REGION Network 13: Check Pressure
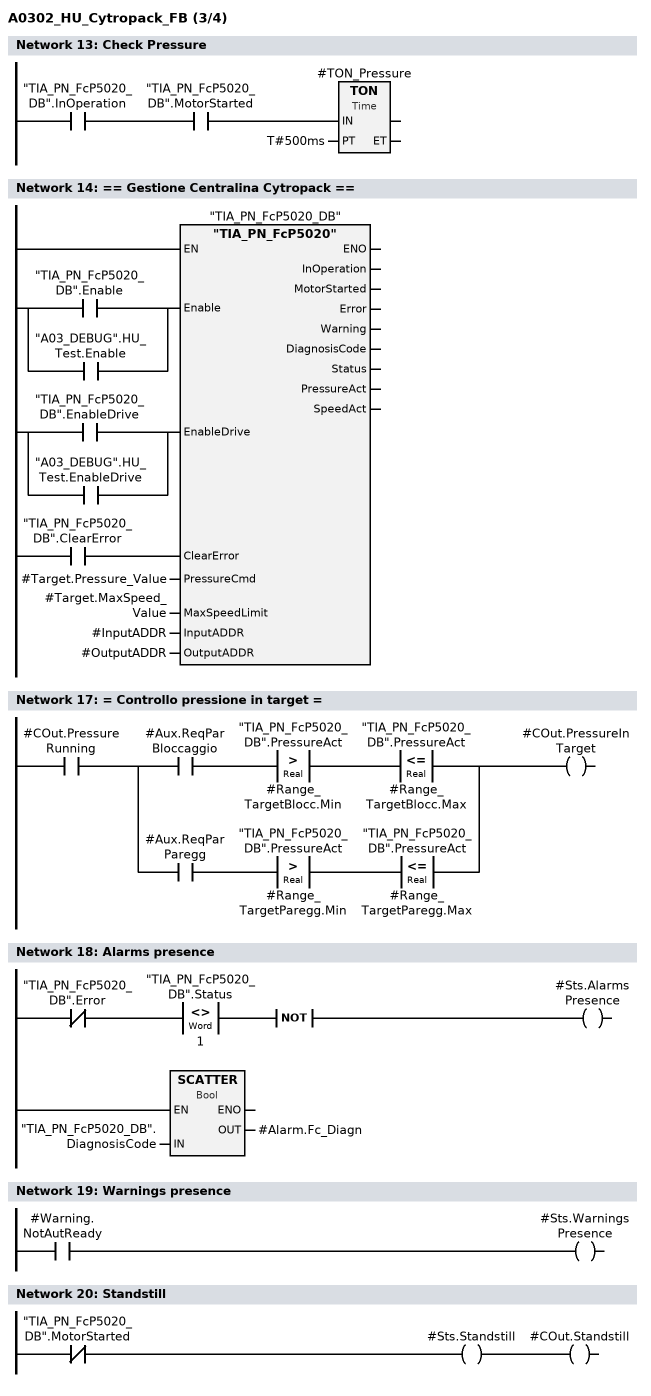
   RUNG wire#powerrail
      Contact( "TIA_PN_FcP5020_DB".InOperation )
      Contact( "TIA_PN_FcP5020_DB".MotorStarted )
      { S7_Templates := "time_type := Time" } #TON_Pressure.TON(pt := T#500ms, et =>)
   END_RUNG
   // the same network as SCL:
   #TON_Pressure.TON(IN := "TIA_PN_FcP5020_DB".InOperation AND "TIA_PN_FcP5020_DB".MotorStarted, PT := T#500ms);
END_REGION

REGION Network 14: == Gestione Centralina Cytropack ==
   RUNG wire#powerrail
      "TIA_PN_FcP5020_DB"(Enable := wire#w1, EnableDrive := wire#w2, ClearError := wire#w3, PressureCmd := #Target.Pressure_Value, MaxSpeedLimit := #Target.MaxSpeed_Value, InputADDR := #InputADDR, OutputADDR := #OutputADDR, InOperation =>, MotorStarted =>, Error =>, Warning =>, DiagnosisCode =>, Status =>, PressureAct =>, SpeedAct =>)
   END_RUNG
   RUNG wire#powerrail
      Contact( "TIA_PN_FcP5020_DB".Enable )
   END_RUNG wire#w1
   RUNG wire#powerrail
      Contact( "A03_DEBUG".HU_Test.Enable )
   END_RUNG wire#w1
   RUNG wire#powerrail
      Contact( "TIA_PN_FcP5020_DB".EnableDrive )
   END_RUNG wire#w2
   RUNG wire#powerrail
      Contact( "A03_DEBUG".HU_Test.EnableDrive )
   END_RUNG wire#w2
   RUNG wire#powerrail
      Contact( "TIA_PN_FcP5020_DB".ClearError )
   END_RUNG wire#w3
   // the same network as SCL:
   "TIA_PN_FcP5020_DB"(Enable := "TIA_PN_FcP5020_DB".Enable OR "A03_DEBUG".HU_Test.Enable,   // "TIA_PN_FcP5020"
                       EnableDrive := "TIA_PN_FcP5020_DB".EnableDrive OR "A03_DEBUG".HU_Test.EnableDrive,
                       ClearError := "TIA_PN_FcP5020_DB".ClearError,
                       PressureCmd := #Target.Pressure_Value,
                       MaxSpeedLimit := #Target.MaxSpeed_Value,
                       InputADDR := #InputADDR,
                       OutputADDR := #OutputADDR);
END_REGION

REGION Network 16: <<< MACHINE STATUS >>>
END_REGION

REGION Network 17: = Controllo pressione in target =
   RUNG wire#powerrail
      Contact( #COut.PressureRunning )
      wire#w1
      Contact( #Aux.ReqParBloccaggio )
      { S7_Templates := "SrcType := Real" } GT_Contact(in1 := "TIA_PN_FcP5020_DB".PressureAct, in2 := #Range_TargetBlocc.Min)
      { S7_Templates := "SrcType := Real" } LE_Contact(in1 := "TIA_PN_FcP5020_DB".PressureAct, in2 := #Range_TargetBlocc.Max)
      wire#w2
      Coil( #COut.PressureInTarget )
   END_RUNG
   RUNG wire#w1
      Contact( #Aux.ReqParParegg )
      { S7_Templates := "SrcType := Real" } GT_Contact(in1 := "TIA_PN_FcP5020_DB".PressureAct, in2 := #Range_TargetParegg.Min)
      { S7_Templates := "SrcType := Real" } LE_Contact(in1 := "TIA_PN_FcP5020_DB".PressureAct, in2 := #Range_TargetParegg.Max)
   END_RUNG wire#w2
   // the same network as SCL:
   #COut.PressureInTarget := #COut.PressureRunning AND ((#Aux.ReqParBloccaggio AND ("TIA_PN_FcP5020_DB".PressureAct > #Range_TargetBlocc.Min) AND ("TIA_PN_FcP5020_DB".PressureAct <= #Range_TargetBlocc.Max)) OR (#Aux.ReqParParegg AND ("TIA_PN_FcP5020_DB".PressureAct > #Range_TargetParegg.Min) AND ("TIA_PN_FcP5020_DB".PressureAct <= #Range_TargetParegg.Max)));
END_REGION

REGION Network 18: Alarms presence
   RUNG wire#powerrail
      I_Contact( "TIA_PN_FcP5020_DB".Error )
      { S7_Templates := "SrcType := Word" } NE_Contact(in1 := "TIA_PN_FcP5020_DB".Status, in2 := 1)
      Not()
      Coil( #Sts.AlarmsPresence )
   END_RUNG
   RUNG wire#powerrail
      { S7_Templates := "[dest_type := Bool, src_type := Word]" } SCATTER(IN := "TIA_PN_FcP5020_DB".DiagnosisCode, OUT => #Alarm.Fc_Diagn)
   END_RUNG
   // the same network as SCL:
   #Sts.AlarmsPresence := NOT (NOT "TIA_PN_FcP5020_DB".Error AND ("TIA_PN_FcP5020_DB".Status <> 1));
   SCATTER(IN := "TIA_PN_FcP5020_DB".DiagnosisCode, OUT => #Alarm.Fc_Diagn);
END_REGION

REGION Network 19: Warnings presence
   RUNG wire#powerrail
      Contact( #Warning.NotAutReady )
      Coil( #Sts.WarningsPresence )
   END_RUNG
   // the same network as SCL:
   #Sts.WarningsPresence := #Warning.NotAutReady;
END_REGION

REGION Network 20: Standstill
   RUNG wire#powerrail
      I_Contact( "TIA_PN_FcP5020_DB".MotorStarted )
      Coil( #Sts.Standstill )
      Coil( #COut.Standstill )
   END_RUNG
   // the same network as SCL:
   #Sts.Standstill := NOT "TIA_PN_FcP5020_DB".MotorStarted;
   #COut.Standstill := NOT "TIA_PN_FcP5020_DB".MotorStarted;
END_REGION

REGION Network 21: Stop for aborting
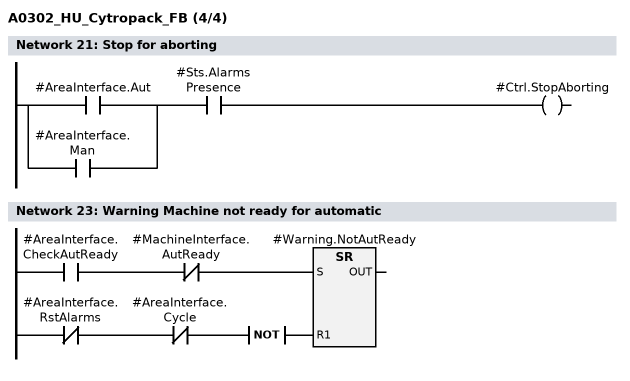
   RUNG wire#powerrail
      Contact( #AreaInterface.Aut )
      wire#w1
      Contact( #Sts.AlarmsPresence )
      Coil( #Ctrl.StopAborting )
   END_RUNG
   RUNG wire#powerrail
      Contact( #AreaInterface.Man )
   END_RUNG wire#w1
   // the same network as SCL:
   #Ctrl.StopAborting := (#AreaInterface.Aut OR #AreaInterface.Man) AND #Sts.AlarmsPresence;
END_REGION

REGION Network 22 (SCL): Collect machine to zone interface

   #MachineInterface.AutReady := #AreaInterface.Aut AND NOT #Sts.AlarmsPresence;
   #MachineInterface.Aborting := #Ctrl.StopAborting;
   #MachineInterface.MotionsStandStill := #TON_NoPendingCmd.Q AND #Sts.Standstill;
   #MachineInterface.AckStopInPhase := #Ctrl.StopInPhase  AND #MachineInterface.MotionsStandStill;
   #MachineInterface.AckStopProgrammed := #Ctrl.StopProgrammed AND #MachineInterface.MotionsStandStill;
   #MachineInterface.AlarmsPresence := #Sts.AlarmsPresence;
   #MachineInterface.WarningPresence := #Sts.WarningsPresence;
END_REGION

REGION Network 23: Warning Machine not ready for automatic
   RUNG wire#powerrail
      Contact( #AreaInterface.CheckAutReady )
      I_Contact( #MachineInterface.AutReady )
      S_SR(operand := #Warning.NotAutReady, r1 := wire#w1)
   END_RUNG
   RUNG wire#powerrail
      I_Contact( #AreaInterface.RstAlarms )
      I_Contact( #AreaInterface.Cycle )
      Not()
   END_RUNG wire#w1
   // the same network as SCL:
   IF #AreaInterface.CheckAutReady AND NOT #MachineInterface.AutReady THEN
       #Warning.NotAutReady := TRUE;   // SR flip-flop
   END_IF;
   IF NOT (NOT #AreaInterface.RstAlarms AND NOT #AreaInterface.Cycle) THEN
       #Warning.NotAutReady := FALSE;
   END_IF;
END_REGION

REGION Network 24 (SCL): Return value variable
   (* LBO TEST
   // Read data from EFC's PROFINET input area
   #iReturnVal := DPRD_DAT(LADDR := #InputADDR, RECORD => #stInputData);
   // Read data failed
   IF (#iReturnVal <> 0) THEN
       #Error := TRUE;
       #bFBErrorDPRD_DPWR := TRUE;
       RETURN;
   END_IF;
   *)
END_REGION
END_FUNCTION_BLOCK

FUNCTION "A0302_Spintore_CALL" : Void   // FC1, LAD
// stored: SetENOAutomatically false
   VAR_TEMP
      Missing_Input : Bool;
      Missing_Output : Bool;
   END_VAR
   VAR CONSTANT
      MISSING : Int;
   END_VAR
BEGIN

REGION Network 1 (SCL): << TRASFERIMENTO stati CIn del blocco >>
   REGION TRASFERIMENTO CIn MANAGER
       "A0302_Spintore".Cin.Manager := "A0302_Manager".COut.SpintoreLong;
       //
       "A0302_Spintore".Cin.SemiAut_Pb := "A0302_Manager".DataIn.SemiAut_Pb;

   END_REGION ;

   REGION TRASFERIMENTO BORDATRICE
       "A0302_Spintore".Cin.Bordatrice.Ax := "A0302_Bordatrice".COut.Ax;
       "A0302_Spintore".Cin.Bordatrice.Sens.FTC_Uscita := "A0302_Bordatrice".IEC_FTC_UscitaBordatrice.FTC_On;
       "A0302_Spintore".Cin.Bordatrice.Perc_Vel := 50.0;
       "A0302_Spintore".Cin.Bordatrice.TargetVel := "A0302_Bordatrice".COut.Ax.ActualVelocity;

   END_REGION ;

   REGION TRASFERIMENTO CIn FERMI P4
       "A0302_Spintore".Cin.P4.Fermi := "A0301_Fermi_P4".COut.Fermi;
   END_REGION ;

   REGION TRASFERIMENTO SPINTORI LATERALI CIn P5
       "A0302_Spintore".Cin.P5.Spintore_Lat.Spin_Lat1 := "A0301_Spintore_Lat".COut.Spin_Lat1;
       "A0302_Spintore".Cin.P5.Spintore_Lat.Spin_Lat2 := "A0301_Spintore_Lat".COut.Spin_Lat2;
       "A0302_Spintore".Cin.P5."En/Dis_SpinLat_2" := "A0301_Spintore_Lat".Sts."En/Dis_SpinLat_2";
       "A0302_Spintore".Cin.P5.QuotaIngombro_SpinLat2 := "PrjConfig_A03".A0301.SpintoreLaterale.QuotaIngombro_SpinLat2;
       "A0302_Spintore".Cin.P5.QuotaIngombro_SpinLat1 := "PrjConfig_A03".A0301.SpintoreLaterale.QuotaIngombro_SpinLat1;

   END_REGION ;

   REGION TRASFERIMENTO CIn TRASPORTO 
       // Trasferimenti status lettura posizioni Trasporto al Cin delle stazioni
       "A0302_Spintore".Cin.Trasporto := "A0301_Trasporto".COut.Ax;
   END_REGION ;
END_REGION

REGION Network 2 (SCL): << TRASFERIMENTO stati DataIn >>
   REGION TRASFERIMENTO #DataIn STATI OPERATION BUTTON STAZIONE SPINTORE LATERALE 
       // PB FERMI VERTICALI
       "A0302_Spintore".DataIn.OP.Rest := "A03_HMI".MB3.Button.A0302.SpintoreLong.OP.Rest;
       "A0302_Spintore".DataIn.OP.Work := "A03_HMI".MB3.Button.A0302.SpintoreLong.OP.Work;
   END_REGION ;

   REGION TRASFERIMENTO STATO LETTURA SENSORI SPINTORE 

       "A0302_Spintore".DataIn.P5.Orz_AnalSens := "A0302_AI_Ammortizatore_Posizionamento";
       "A0302_Spintore".DataIn.P5.FTC_FuoriIngombro_A0301 := "A0302_Bordatrice_Banco_4_Lato_1_Phc_AtEntry";

   END_REGION ;
END_REGION

REGION Network 3: << DataIn Ax - Asse Spintore pezzo >>
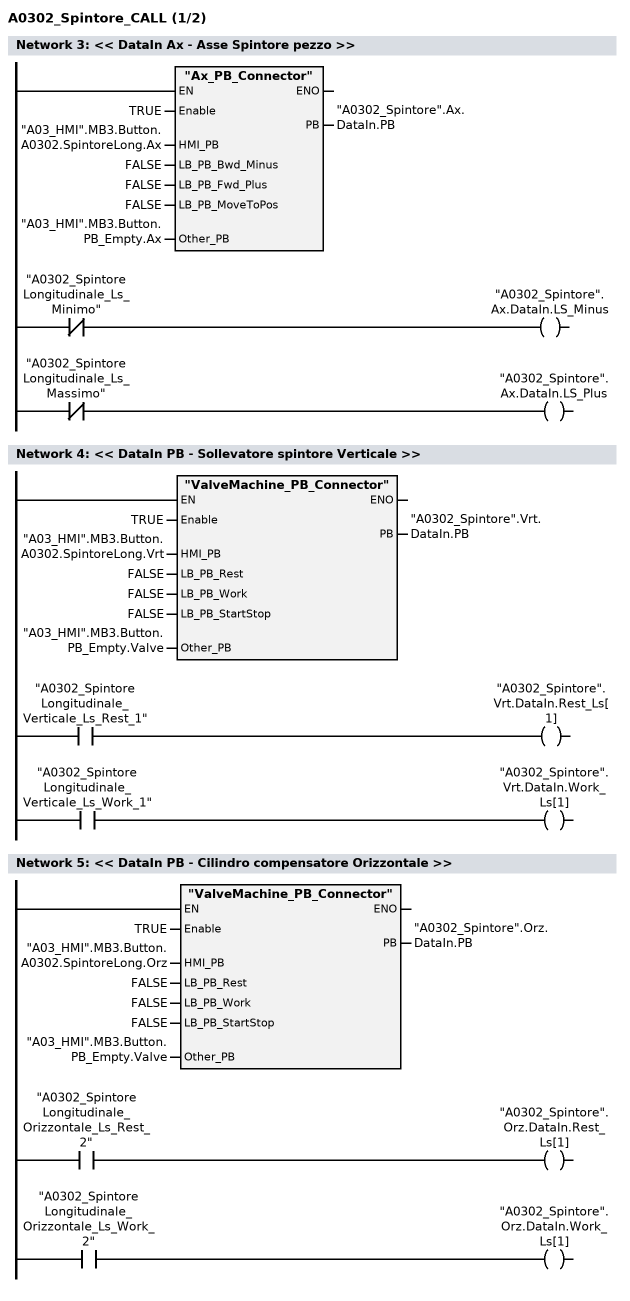
   RUNG wire#powerrail
      "Ax_PB_Connector"(Enable := TRUE, HMI_PB := "A03_HMI".MB3.Button.A0302.SpintoreLong.Ax, LB_PB_Bwd_Minus := FALSE, LB_PB_Fwd_Plus := FALSE, LB_PB_MoveToPos := FALSE, Other_PB := "A03_HMI".MB3.Button.PB_Empty.Ax, PB => "A0302_Spintore".Ax.DataIn.PB)
   END_RUNG
   RUNG wire#powerrail
      I_Contact( "A0302_SpintoreLongitudinale_Ls_Minimo" )
      Coil( "A0302_Spintore".Ax.DataIn.LS_Minus )
   END_RUNG
   RUNG wire#powerrail
      I_Contact( "A0302_SpintoreLongitudinale_Ls_Massimo" )
      Coil( "A0302_Spintore".Ax.DataIn.LS_Plus )
   END_RUNG
   // the same network as SCL:
   "Ax_PB_Connector"(Enable := TRUE,
                     HMI_PB := "A03_HMI".MB3.Button.A0302.SpintoreLong.Ax,
                     LB_PB_Bwd_Minus := FALSE,
                     LB_PB_Fwd_Plus := FALSE,
                     LB_PB_MoveToPos := FALSE,
                     Other_PB := "A03_HMI".MB3.Button.PB_Empty.Ax,
                     PB => "A0302_Spintore".Ax.DataIn.PB);
   "A0302_Spintore".Ax.DataIn.LS_Minus := NOT "A0302_SpintoreLongitudinale_Ls_Minimo";
   "A0302_Spintore".Ax.DataIn.LS_Plus := NOT "A0302_SpintoreLongitudinale_Ls_Massimo";
END_REGION

REGION Network 4: << DataIn PB - Sollevatore spintore Verticale >>
   RUNG wire#powerrail
      "ValveMachine_PB_Connector"(Enable := TRUE, HMI_PB := "A03_HMI".MB3.Button.A0302.SpintoreLong.Vrt, LB_PB_Rest := FALSE, LB_PB_Work := FALSE, LB_PB_StartStop := FALSE, Other_PB := "A03_HMI".MB3.Button.PB_Empty.Valve, PB => "A0302_Spintore".Vrt.DataIn.PB)
   END_RUNG
   RUNG wire#powerrail
      Contact( "A0302_SpintoreLongitudinale_Verticale_Ls_Rest_1" )
      Coil( "A0302_Spintore".Vrt.DataIn.Rest_Ls[1] )
   END_RUNG
   RUNG wire#powerrail
      Contact( "A0302_SpintoreLongitudinale_Verticale_Ls_Work_1" )
      Coil( "A0302_Spintore".Vrt.DataIn.Work_Ls[1] )
   END_RUNG
   // the same network as SCL:
   "ValveMachine_PB_Connector"(Enable := TRUE,
                           HMI_PB := "A03_HMI".MB3.Button.A0302.SpintoreLong.Vrt,
                           LB_PB_Rest := FALSE,
                           LB_PB_Work := FALSE,
                           LB_PB_StartStop := FALSE,
                           Other_PB := "A03_HMI".MB3.Button.PB_Empty.Valve,
                           PB => "A0302_Spintore".Vrt.DataIn.PB);
   "A0302_Spintore".Vrt.DataIn.Rest_Ls[1] := "A0302_SpintoreLongitudinale_Verticale_Ls_Rest_1";
   "A0302_Spintore".Vrt.DataIn.Work_Ls[1] := "A0302_SpintoreLongitudinale_Verticale_Ls_Work_1";
END_REGION

REGION Network 5: << DataIn PB - Cilindro compensatore Orizzontale >>
   RUNG wire#powerrail
      "ValveMachine_PB_Connector"(Enable := TRUE, HMI_PB := "A03_HMI".MB3.Button.A0302.SpintoreLong.Orz, LB_PB_Rest := FALSE, LB_PB_Work := FALSE, LB_PB_StartStop := FALSE, Other_PB := "A03_HMI".MB3.Button.PB_Empty.Valve, PB => "A0302_Spintore".Orz.DataIn.PB)
   END_RUNG
   RUNG wire#powerrail
      Contact( "A0302_SpintoreLongitudinale_Orizzontale_Ls_Rest_2" )
      Coil( "A0302_Spintore".Orz.DataIn.Rest_Ls[1] )
   END_RUNG
   RUNG wire#powerrail
      Contact( "A0302_SpintoreLongitudinale_Orizzontale_Ls_Work_2" )
      Coil( "A0302_Spintore".Orz.DataIn.Work_Ls[1] )
   END_RUNG
   // the same network as SCL:
   "ValveMachine_PB_Connector"(Enable := TRUE,
                           HMI_PB := "A03_HMI".MB3.Button.A0302.SpintoreLong.Orz,
                           LB_PB_Rest := FALSE,
                           LB_PB_Work := FALSE,
                           LB_PB_StartStop := FALSE,
                           Other_PB := "A03_HMI".MB3.Button.PB_Empty.Valve,
                           PB => "A0302_Spintore".Orz.DataIn.PB);
   "A0302_Spintore".Orz.DataIn.Rest_Ls[1] := "A0302_SpintoreLongitudinale_Orizzontale_Ls_Rest_2";
   "A0302_Spintore".Orz.DataIn.Work_Ls[1] := "A0302_SpintoreLongitudinale_Orizzontale_Ls_Work_2";
END_REGION

REGION Network 6 (SCL): DSI
   //
   "A0302_Spintore".DSI_Feed := "F_DB".DSI_Spintore;
   "A0302_Spintore".DSI_Valve := "F_DB".DSI_V_Air_A0301_A0302;
END_REGION

REGION Network 7 (SCL): HW
   "A0302_Spintore".HWID_Ax_TEL111 := "HW_Const_Values".CU5_PN_1560A1_2_Standard_telegram_1_2;
END_REGION

REGION Network 8 (SCL): Drive
   //
   "A0302_Spintore".Drive.Infeed_ON := "Areas_ITF".AG.Infeed_Running;
   "A0302_Spintore".Drive.AccessPoint :=  "HW_Const_Values".CU5_PN_600A1_ModuleAccessPoint;
   "A0302_Spintore".Drive.AxisID := "CU5_ID_6_1560A1_2_1600M1";
   "A0302_Spintore".Drive.TokenChain := "TOKENCHAIN_CU5";
END_REGION

REGION Network 9: [Spintore Longitudinale] - Machine Call
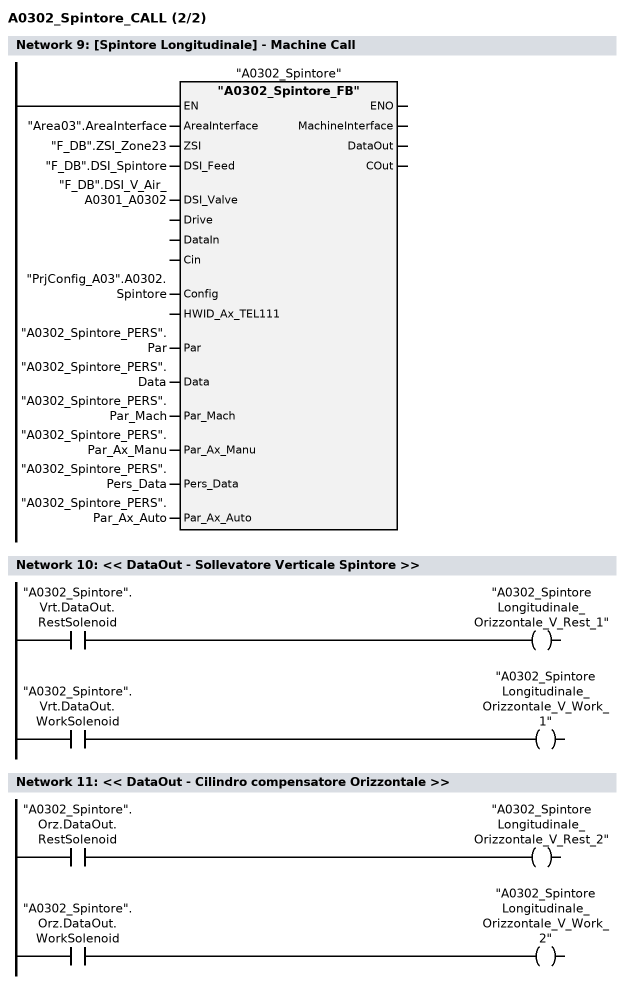
   RUNG wire#powerrail
      "A0302_Spintore"(AreaInterface := "Area03".AreaInterface, ZSI := "F_DB".ZSI_Zone23, DSI_Feed := "F_DB".DSI_Spintore, DSI_Valve := "F_DB".DSI_V_Air_A0301_A0302, Drive :=, DataIn :=, Cin :=, Config := "PrjConfig_A03".A0302.Spintore, HWID_Ax_TEL111 :=, Par := "A0302_Spintore_PERS".Par, Data := "A0302_Spintore_PERS".Data, Par_Mach := "A0302_Spintore_PERS".Par_Mach, Par_Ax_Manu := "A0302_Spintore_PERS".Par_Ax_Manu, Pers_Data := "A0302_Spintore_PERS".Pers_Data, Par_Ax_Auto := "A0302_Spintore_PERS".Par_Ax_Auto, MachineInterface =>, DataOut =>, COut =>)
   END_RUNG
   // the same network as SCL:
   "A0302_Spintore"(AreaInterface := "Area03".AreaInterface,   // "A0302_Spintore_FB"
                    ZSI := "F_DB".ZSI_Zone23,
                    DSI_Feed := "F_DB".DSI_Spintore,
                    DSI_Valve := "F_DB".DSI_V_Air_A0301_A0302,
                    Config := "PrjConfig_A03".A0302.Spintore,
                    Par := "A0302_Spintore_PERS".Par,
                    Data := "A0302_Spintore_PERS".Data,
                    Par_Mach := "A0302_Spintore_PERS".Par_Mach,
                    Par_Ax_Manu := "A0302_Spintore_PERS".Par_Ax_Manu,
                    Pers_Data := "A0302_Spintore_PERS".Pers_Data,
                    Par_Ax_Auto := "A0302_Spintore_PERS".Par_Ax_Auto);
END_REGION

REGION Network 10: << DataOut - Sollevatore Verticale Spintore >>
   RUNG wire#powerrail
      Contact( "A0302_Spintore".Vrt.DataOut.RestSolenoid )
      Coil( "A0302_SpintoreLongitudinale_Orizzontale_V_Rest_1" )
   END_RUNG
   RUNG wire#powerrail
      Contact( "A0302_Spintore".Vrt.DataOut.WorkSolenoid )
      Coil( "A0302_SpintoreLongitudinale_Orizzontale_V_Work_1" )
   END_RUNG
   // the same network as SCL:
   "A0302_SpintoreLongitudinale_Orizzontale_V_Rest_1" := "A0302_Spintore".Vrt.DataOut.RestSolenoid;
   "A0302_SpintoreLongitudinale_Orizzontale_V_Work_1" := "A0302_Spintore".Vrt.DataOut.WorkSolenoid;
END_REGION

REGION Network 11: << DataOut - Cilindro compensatore Orizzontale >>
   RUNG wire#powerrail
      Contact( "A0302_Spintore".Orz.DataOut.RestSolenoid )
      Coil( "A0302_SpintoreLongitudinale_Orizzontale_V_Rest_2" )
   END_RUNG
   RUNG wire#powerrail
      Contact( "A0302_Spintore".Orz.DataOut.WorkSolenoid )
      Coil( "A0302_SpintoreLongitudinale_Orizzontale_V_Work_2" )
   END_RUNG
   // the same network as SCL:
   "A0302_SpintoreLongitudinale_Orizzontale_V_Rest_2" := "A0302_Spintore".Orz.DataOut.RestSolenoid;
   "A0302_SpintoreLongitudinale_Orizzontale_V_Work_2" := "A0302_Spintore".Orz.DataOut.WorkSolenoid;
END_REGION
END_FUNCTION

FUNCTION_BLOCK "A0302_Spintore_FB"   // FB91, LAD
// stored: MemoryReserve 100, SetENOAutomatically false
   VAR_INPUT
      AreaInterface : "AreaInterface";
      ZSI : "udt_ZoneSafetyInterface";
      DSI_Feed : "udt_DeviceSafetyInterface";
      DSI_Valve : "udt_DeviceSafetyInterface";
      Drive : "TAx_DriveInterface";
      DataIn : Struct
         OP : "OP_PB";
         P5 { ExternalAccessible := 'False'; ExternalVisible := 'False'; ExternalWritable := 'False'} : Struct
            Orz_AnalSens : Int;
            FTC_FuoriIngombro_A0301 : Bool;   // FTC fuori ingombro lato bordatrice
         END_STRUCT;
      END_STRUCT;
      Cin : Struct
         Manager { ExternalWritable := 'False'} : Struct
            EnableStopDoorOpeningReq : Bool;
            EnableStopInPhase : Bool;
            EnableStopProgrammed : Bool;
            Control_ON : Bool;
            REST_Req : Bool;
            WORK_Req : Bool;
            Rest : Bool;
            Work : Bool;
         END_STRUCT;
         SemiAut_Pb { ExternalAccessible := 'False'; ExternalVisible := 'False'; ExternalWritable := 'False'} : Bool;
         P4 { ExternalWritable := 'False'} : Struct
            Fermi : "ValveMachine_COut";
         END_STRUCT;
         P5 { ExternalWritable := 'False'} : Struct
            "En/Dis_SpinLat_2" : Bool;   // 1=Enable / 0=Disable
            QuotaIngombro_SpinLat2 : Real;
            QuotaIngombro_SpinLat1 : Real;
            Spintore_Lat : Struct
               Spin_Lat1 : Struct
                  Standstill : Bool;
                  Rest_CheckNext : Bool;
                  Work_CheckNext : Bool;
                  Rest : Bool;
                  Work : Bool;
               END_STRUCT;
               Spin_Lat2 : Struct
                  Standstill : Bool;
                  Rest_CheckNext : Bool;
                  Work_CheckNext : Bool;
                  Rest : Bool;
                  Work : Bool;
               END_STRUCT;
               Vrt_1 : "ValveMachine_COut";
               Orz_1 : "ValveMachine_COut";
               Vrt_2 : "ValveMachine_COut";
               Orz_2 : "ValveMachine_COut";
               Sollevatori : "ValveMachine_COut";
            END_STRUCT;
         END_STRUCT;
         Trasporto { ExternalAccessible := 'False'; ExternalVisible := 'False'; ExternalWritable := 'False'} : "SpeedMachine_COut";
         Bordatrice : Struct   // *************************
            Ax : "Positioning_EPOS_Machine_COut";
            TargetVel : LReal;
            Perc_Vel : LReal;
            Sens : Struct
               FTC_Uscita : Bool;
            END_STRUCT;
         END_STRUCT;
      END_STRUCT;
      Config : Struct
         Ax : "Positioning_EPOS_Machine_Config_NEW";
         Vrt : "ValveMachine_Config";
         Orz : "ValveMachine_Config";
         SpintoreLat : Struct
            QuotaIngombro_SpinLat2 : Real := 2705.0;
            QuotaIngombro_SpinLat1 : Real := 4777.0;
         END_STRUCT;
         Bordatrice : Struct
            QuotaIngresso : Real := 600.0;
         END_STRUCT;
         DelayMissingCondition : Time;
      END_STRUCT;
      HWID_Ax_TEL111 : HW_SUBMODULE;
   END_VAR
   VAR_OUTPUT
      MachineInterface : "MachineInterface";
      DataOut : "Positioning_EPOS_Machine_DataOut";
      COut : Struct
         Ax_Sts : Struct
            PosAttesa_Reached : Bool;
            PosFineSpinta_Reached : Bool;
         END_STRUCT;
         Ax : "Positioning_EPOS_Machine_COut";
         Spintore : "ValveMachine_COut";
         Vrt : "ValveMachine_COut";
         Orz : "ValveMachine_COut";
      END_STRUCT;
   END_VAR
   VAR_IN_OUT
      Par : Struct
         Sens : "Analogic_SensorManagement_Par";
      END_STRUCT;
      Data : Struct
         Sens : "Analogic_SensorManagement_Data";
         HMI : "HMI_Preset";
         Ax_Pos : "A0301_Mach_Ax_Pos_Data";
      END_STRUCT;
      Par_Mach : "A0301_Mach_Sens_Par";
      Par_Ax_Manu : "Positioning_EPOS_Machine_Par";
      Pers_Data : Struct
         EncoderAbsolute_Preset_OK : Bool;
         Persistent_ActualPosition : LReal;
      END_STRUCT;
      Par_Ax_Auto : "A0301_Mach_Speed_Par";
   END_VAR
   VAR
      Alarm : Struct
         Ax : "Positioning_EPOS_Machine_Alr";
         Ax_NeedPreset { S7_SetPoint := 'True'} : Bool;
         Vrt : "ValveAlr";
         Orz : "ValveAlr";
         Orz_AnalSens_Issue : Bool;
         Orz_AnalSens_Compressed : Bool;
      END_STRUCT;
      Warning : Struct
         Ax : "Positioning_EPOS_Machine_Wng";
         Vrt : "ValveMachine_Wng";
         Orz { S7_SetPoint := 'True'} : "ValveMachine_Wng";
         Orz_AnalSens { S7_SetPoint := 'True'} : "Analogic_SensorManagement_Warning";
         OP_REST_MissingCnd : Bool;   // Mancanza comando arresto
         OP_WORK_MissingCnd : Bool;   // Mancanza consenso lavoro
      END_STRUCT;
      Sts : Struct
         ReadyForMove : Bool;   // Pronto al movimento
         OP_CanMoveFreely : Bool;
         OP_Ax_Rest_Cnd : Bool;
         OP_Ax_Work_Cnd : Bool;
         OP_Spin_Rest_Cnd : Bool;
         OP_Spin_Work_Cnd : Bool;
         A0301_Beam_BLean : Real;
         A0302_Beam_BLean : Real;
         Vrt_Work_ExtEnable : Bool;
         Orz_Work_ExtEnable : Bool;
      END_STRUCT;
      Ctrl : Struct
         SpinVrtOrz : Struct
            OP_Rest_Man : Bool;
            OP_Work_Man : Bool;
            OP_Rest_Aut : Bool;
            OP_Work_Aut : Bool;
            OP_Rest : Bool;
            OP_Work : Bool;
         END_STRUCT;
         Ax : Struct
            OP_Rest_Man : Bool;
            OP_Work_Man : Bool;
            OP_Rest_Aut : Bool;
            OP_Work_Aut : Bool;
            OP_Rest : Bool;
            OP_Work : Bool;
            Vel : LReal;
            VelMax : Real;
            Dec : LReal;
         END_STRUCT;
      END_STRUCT;
      HMI : Struct
         Ax : "AnalogSens_HmiData";
         Orz_AnalSens_PB_Preset { ExternalAccessible := 'False'; ExternalVisible := 'False'; ExternalWritable := 'False'} : Bool;   // Pulsante Preset value
         Orz_AnalSens_Preset_Value : LReal;
      END_STRUCT;
      Ax { S7_SetPoint := 'True'} : "Positioning_EPOS_Machine_FB_NEW";   // Spintore longitudinale
      Vrt { S7_SetPoint := 'True'} : "ValveMachine_FB";   // Sollevatore verticale
      Orz { S7_SetPoint := 'True'} : "ValveMachine_FB";   // Compensatore orizzontale
      Orz_AnalSens { S7_SetPoint := 'True'} : "Analogic_SensorManagement";
      ValueBLeanOvr : Array[1..15] of Real;
      IEC : Struct
         TON_DelayFTC_Ingombro_A0301 : IEC_TIMER;
         TOF_DelayFTC_Ingombro_A0301 { S7_SetPoint := 'True'} : IEC_TIMER;
         FTC_On { S7_SetPoint := 'True'} : Bool;
      END_STRUCT;
      AUX : Struct
         OP_Rest_PB : Bool;
         OP_Work_PB : Bool;
      END_STRUCT;
      TON_OP_REST_MissingCnd { S7_SetPoint := 'True'} : TON_TIME;
      TON_OP_WORK_MissingCnd { S7_SetPoint := 'True'} : TON_TIME;
      BTrk_Item : Struct
         BLean : Real;
         O_ID : DInt;
      END_STRUCT;
   END_VAR
   VAR_TEMP
      i : Int;
      DecMax : LReal;
      Orz_SpazioSafe : LReal;
      Calcoli : Struct
         SUB_SpinLat2 : LReal;
         SUB_SpinLat1 : LReal;
         Pos_Target_2 : LReal;
         Pos_Target_1 : LReal;
         Ax_Target : LReal;
      END_STRUCT;
      PE : Struct
         OP_Rest_PB : Bool;
         OP_Work_PB : Bool;
      END_STRUCT;
      BTrk_GetData_A0302 : Struct
         indx : Int;   // Se trovato tra i TODO / ENDING / OUT questo è l'indice dove sono stati prelevati i dati
         Sts : Int;   // 0 = Non Trovato; 0 = ACT; 1 = TODO; 2=ENDING; 3 = OUT
         Item : "Prod_Item_small";
      END_STRUCT;
      BTrk_GetData_A0301 : Struct
         indx : Int;   // Se trovato tra i TODO / ENDING / OUT questo è l'indice dove sono stati prelevati i dati
         Sts : Int;   // 0 = Non Trovato; 0 = ACT; 1 = TODO; 2=ENDING; 3 = OUT
         Item : "Prod_Item_small";
      END_STRUCT;
      Stop_Ax_SpinLong : Bool;
      GetData_A0301_B : Bool;
      GetData_A0302_In : Bool;
   END_VAR
   VAR CONSTANT
      Offset_SpinLong_To_SpinLat2 : Real;   // Offset calcolato da quota ingombro Spintore Laterale2 per bloccare Spintore Longitudinale e allarme se SpinLat2 alto
      Offset_SpinLong_To_SpinLat1 : Real;   // Offset calcolato da quota ingombro Spintore Laterale1 per bloccare Spintore Longitudinale e allarme se SpinLat1 alto
   END_VAR
   // Orz_AnalSens.Filter.Tau := T#10ms;
   VAR_TEMP   // added for the SCL form of the ladder/FBD networks
      _w1 : Bool;
      _w2 : Bool;
      _w3 : Bool;
      _w4 : Bool;
      _w5 : Bool;
      _w6 : Bool;
   END_VAR
BEGIN

REGION Network 1 (SCL): Reset allarmi
   IF #AreaInterface.RstAlarms THEN
       #Alarm.Orz_AnalSens_Issue := FALSE;
       #Warning.Orz_AnalSens.SignalError := FALSE;
   END_IF;
END_REGION

REGION Network 2: <+>
END_REGION

REGION Network 4: CONTROLLO MES lunghezza Beams
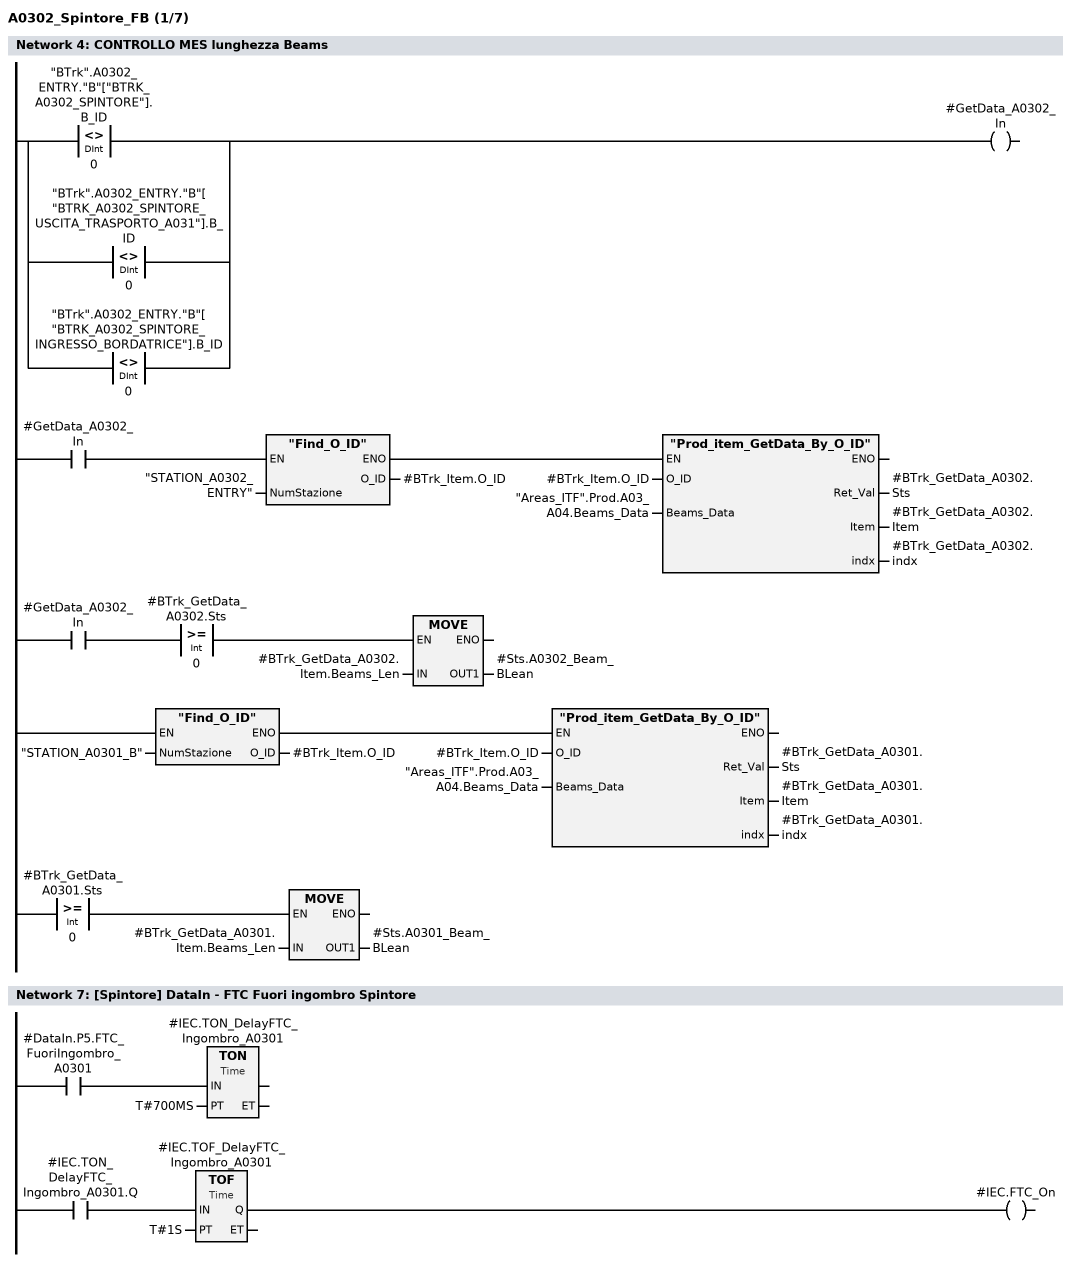
   RUNG wire#powerrail
      { S7_Templates := "SrcType := DInt" } NE_Contact(in1 := "BTrk".A0302_ENTRY."B"["BTRK_A0302_SPINTORE"].B_ID, in2 := 0)
      wire#w1
      Coil( #GetData_A0302_In )
   END_RUNG
   RUNG wire#powerrail
      { S7_Templates := "SrcType := DInt" } NE_Contact(in1 := "BTrk".A0302_ENTRY."B"["BTRK_A0302_SPINTORE_USCITA_TRASPORTO_A031"].B_ID, in2 := 0)
   END_RUNG wire#w1
   RUNG wire#powerrail
      { S7_Templates := "SrcType := DInt" } NE_Contact(in1 := "BTrk".A0302_ENTRY."B"["BTRK_A0302_SPINTORE_INGRESSO_BORDATRICE"].B_ID, in2 := 0)
   END_RUNG wire#w1
   RUNG wire#powerrail
      Contact( #GetData_A0302_In )
      "Find_O_ID"(NumStazione := "STATION_A0302_ENTRY", O_ID => #BTrk_Item.O_ID)
      "Prod_item_GetData_By_O_ID"(O_ID := #BTrk_Item.O_ID, Beams_Data := "Areas_ITF".Prod.A03_A04.Beams_Data, Ret_Val => #BTrk_GetData_A0302.Sts, Item => #BTrk_GetData_A0302.Item, indx => #BTrk_GetData_A0302.indx)
   END_RUNG
   RUNG wire#powerrail
      Contact( #GetData_A0302_In )
      { S7_Templates := "SrcType := Int" } GE_Contact(in1 := #BTrk_GetData_A0302.Sts, in2 := 0)
      Move(in := #BTrk_GetData_A0302.Item.Beams_Len, out1 => #Sts.A0302_Beam_BLean)
   END_RUNG
   RUNG wire#powerrail
      "Find_O_ID"(NumStazione := "STATION_A0301_B", O_ID => #BTrk_Item.O_ID)
      "Prod_item_GetData_By_O_ID"(O_ID := #BTrk_Item.O_ID, Beams_Data := "Areas_ITF".Prod.A03_A04.Beams_Data, Ret_Val => #BTrk_GetData_A0301.Sts, Item => #BTrk_GetData_A0301.Item, indx => #BTrk_GetData_A0301.indx)
   END_RUNG
   RUNG wire#powerrail
      { S7_Templates := "SrcType := Int" } GE_Contact(in1 := #BTrk_GetData_A0301.Sts, in2 := 0)
      Move(in := #BTrk_GetData_A0301.Item.Beams_Len, out1 => #Sts.A0301_Beam_BLean)
   END_RUNG
   // the same network as SCL:
   #GetData_A0302_In := ("BTrk".A0302_ENTRY."B"["BTRK_A0302_SPINTORE"].B_ID <> 0) OR ("BTrk".A0302_ENTRY."B"["BTRK_A0302_SPINTORE_USCITA_TRASPORTO_A031"].B_ID <> 0) OR ("BTrk".A0302_ENTRY."B"["BTRK_A0302_SPINTORE_INGRESSO_BORDATRICE"].B_ID <> 0);
   "Find_O_ID"(EN := #GetData_A0302_In,
               NumStazione := "STATION_A0302_ENTRY",
               O_ID => #BTrk_Item.O_ID,
               ENO => #_w1);
   IF #_w1 THEN
       #BTrk_GetData_A0302.Sts := "Prod_item_GetData_By_O_ID"(O_ID := #BTrk_Item.O_ID,
                               Beams_Data := "Areas_ITF".Prod.A03_A04.Beams_Data,
                               Item => #BTrk_GetData_A0302.Item,
                               indx => #BTrk_GetData_A0302.indx);
   END_IF;
   IF #GetData_A0302_In AND (#BTrk_GetData_A0302.Sts >= 0) THEN
       #Sts.A0302_Beam_BLean := #BTrk_GetData_A0302.Item.Beams_Len;
   END_IF;
   "Find_O_ID"(NumStazione := "STATION_A0301_B", O_ID => #BTrk_Item.O_ID, ENO => #_w2);
   IF #_w2 THEN
       #BTrk_GetData_A0301.Sts := "Prod_item_GetData_By_O_ID"(O_ID := #BTrk_Item.O_ID,
                               Beams_Data := "Areas_ITF".Prod.A03_A04.Beams_Data,
                               Item => #BTrk_GetData_A0301.Item,
                               indx => #BTrk_GetData_A0301.indx);
   END_IF;
   IF #BTrk_GetData_A0301.Sts >= 0 THEN #Sts.A0301_Beam_BLean := #BTrk_GetData_A0301.Item.Beams_Len; END_IF;
END_REGION

REGION Network 5 (SCL): CALCOLI - Posizioni Attesa / Spinta per lavoro Spintore

   #BTrk_GetData_A0302.Item.O_ID := #BTrk_GetData_A0302.Item.O_ID;
   #BTrk_Item.BLean:=#BTrk_GetData_A0302.Item.Beams_Len;
   // ***********************************************************************************************************
   // 
   REGION POSIZIONE ATTESA PEZZO IN ENTRATA

       // Se ho una misura traking vado in posizionamento calcolando la misura del Beams più alta + Offset sennò vado indietro fino a pos. minima
       IF #Sts.A0301_Beam_BLean <> 0 THEN
           #Data.Ax_Pos.PosAttesa := (#Ax.COut.MaxPosition -#Sts.A0301_Beam_BLean) - (#Data.Ax_Pos.OffsetPosAttesa - #Config.Bordatrice.QuotaIngresso);
       ELSIF #Sts.OP_CanMoveFreely THEN
           #BTrk_Item.BLean := 0;
           #Data.Ax_Pos.PosAttesa := ( #Ax.COut.MinPosition) + #Data.Ax_Pos.OffsetPosAttesa;
       END_IF;

   END_REGION ;
   //
   // ***********************************************************************************************************
   // 
   REGION POSIZIONE FINE SPINTA PEZZO IN USCITA

       // CALCOLO Pos.Fine Spinta Target finale
       IF #Sts.A0302_Beam_BLean <> 0 THEN
           #Data.Ax_Pos.PosFineSpinta := (#Ax.COut.MaxPosition - #Sts.A0302_Beam_BLean) + (#Config.Bordatrice.QuotaIngresso);
       ELSIF #BTrk_Item.BLean = 0 THEN
           #Data.Ax_Pos.PosFineSpinta := (#Ax.COut.MaxPosition - #Data.Ax_Pos.OffsetPosAttesa);
       END_IF;

       (*
       // CALCOLO differenza tra Pos.Attesa e Quota ingombro Spintore laterale 2 SE incluso 
       IF #Cin.P5."En/Dis_SpinLat_2"
           AND #Ax.COut.ActualPosition < (#Config.SpintoreLat.QuotaIngombro_SpinLat2 +  #Config.SpintoreLat.OffsetPosAttesa) THEN
           #Calcoli.SUB_SpinLat2 :=((#Data.Ax_Pos.PosAttesa) + (#Config.SpintoreLat.QuotaIngombro_SpinLat2));
       END_IF;

       // CALCOLO differenza tra Pos.Attesa e Quota ingombro Spintore laterale 1 
       IF #Ax.COut.ActualPosition > #Config.SpintoreLat.QuotaIngombro_SpinLat1 THEN
           #Calcoli.SUB_SpinLat1 :=((#Data.Ax_Pos.PosAttesa) + (#Config.SpintoreLat.QuotaIngombro_SpinLat1));
       END_IF;

       // CALCOLI Posizioni Target SPINTORI LATERALI
       #Calcoli.Pos_Target_2 := (#Data.Ax_Pos.PosAttesa) + (#Calcoli.SUB_SpinLat2);
       #Calcoli.Pos_Target_1 := (#Data.Ax_Pos.PosAttesa) + (#Calcoli.SUB_SpinLat1);

       // SPINTORE LATERALE 1&2 - AX - POS. Target
       IF #Cin.P5."En/Dis_SpinLat_2"
           AND #Data.Ax_Pos.PosFineSpinta >= #Calcoli.Pos_Target_2 THEN
           #Calcoli.Ax_Target := #Calcoli.Pos_Target_2;
       ELSIF #Data.Ax_Pos.PosFineSpinta >= #Calcoli.Pos_Target_1
           AND #Ax.COut.ActualPosition < (-#Config.SpintoreLat.QuotaIngombro_SpinLat2) THEN
           #Calcoli.Ax_Target := #Calcoli.Pos_Target_1;
       ELSIF #Ax.#COut.ActualPosition < (-#Config.SpintoreLat.QuotaIngombro_SpinLat1) THEN
           #Calcoli.Ax_Target := #Data.Ax_Pos.PosFineSpinta;
       END_IF;
       *)

   END_REGION ;
   //
   // ***********************************************************************************************************
END_REGION

REGION Network 6: <+>
END_REGION

REGION Network 7: [Spintore] DataIn - FTC Fuori ingombro Spintore
   RUNG wire#powerrail
      Contact( #DataIn.P5.FTC_FuoriIngombro_A0301 )
      { S7_Templates := "time_type := Time" } #IEC.TON_DelayFTC_Ingombro_A0301.TON(pt := T#700MS, et =>)
   END_RUNG
   RUNG wire#powerrail
      Contact( #IEC.TON_DelayFTC_Ingombro_A0301.Q )
      { S7_Templates := "time_type := Time" } #IEC.TOF_DelayFTC_Ingombro_A0301.TOF(pt := T#1S, et =>)
      Coil( #IEC.FTC_On )
   END_RUNG
   // the same network as SCL:
   #IEC.TON_DelayFTC_Ingombro_A0301.TON(IN := #DataIn.P5.FTC_FuoriIngombro_A0301, PT := T#700MS);
   #IEC.TOF_DelayFTC_Ingombro_A0301.TOF(IN := #IEC.TON_DelayFTC_Ingombro_A0301.Q, PT := T#1S);
   #IEC.FTC_On := #IEC.TOF_DelayFTC_Ingombro_A0301.Q;
END_REGION

REGION Network 8: <+>
END_REGION

REGION Network 9: Operazione può muoversi liberamente perchè non sposta nessun BEAM
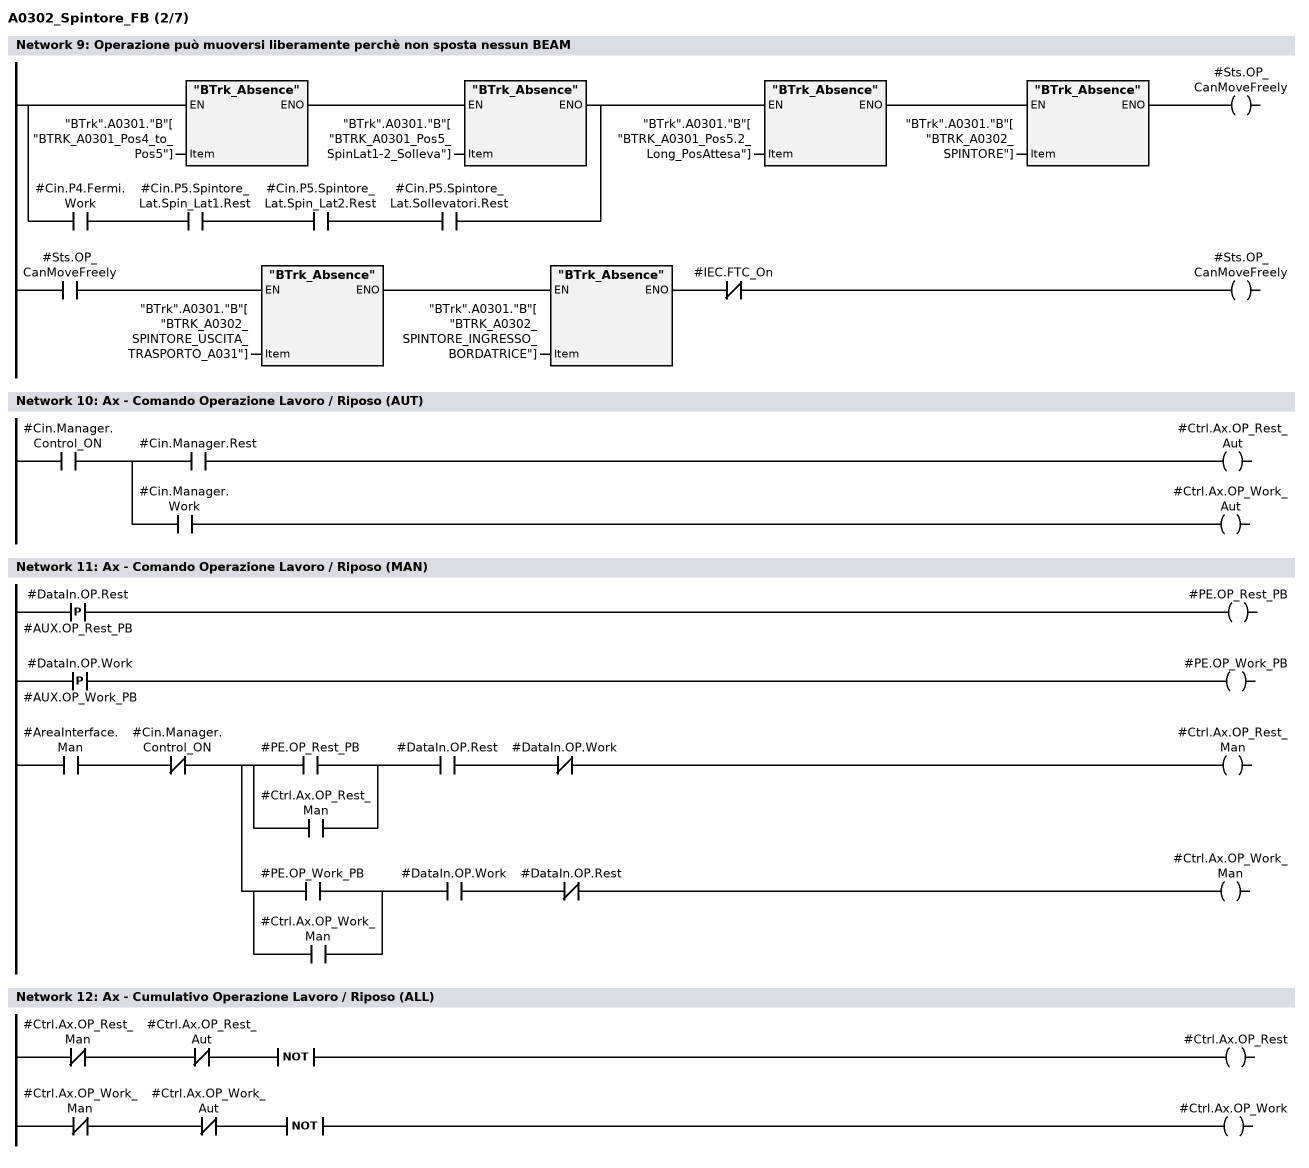
   RUNG wire#powerrail
      "BTrk_Absence"(Item := "BTrk".A0301."B"["BTRK_A0301_Pos4_to_Pos5"])
      "BTrk_Absence"(Item := "BTrk".A0301."B"["BTRK_A0301_Pos5_SpinLat1-2_Solleva"])
      wire#w1
      "BTrk_Absence"(Item := "BTrk".A0301."B"["BTRK_A0301_Pos5.2_Long_PosAttesa"])
      "BTrk_Absence"(Item := "BTrk".A0301."B"["BTRK_A0302_SPINTORE"])
      Coil( #Sts.OP_CanMoveFreely )
   END_RUNG
   RUNG wire#powerrail
      Contact( #Cin.P4.Fermi.Work )
      Contact( #Cin.P5.Spintore_Lat.Spin_Lat1.Rest )
      Contact( #Cin.P5.Spintore_Lat.Spin_Lat2.Rest )
      Contact( #Cin.P5.Spintore_Lat.Sollevatori.Rest )
   END_RUNG wire#w1
   RUNG wire#powerrail
      Contact( #Sts.OP_CanMoveFreely )
      "BTrk_Absence"(Item := "BTrk".A0301."B"["BTRK_A0302_SPINTORE_USCITA_TRASPORTO_A031"])
      "BTrk_Absence"(Item := "BTrk".A0301."B"["BTRK_A0302_SPINTORE_INGRESSO_BORDATRICE"])
      I_Contact( #IEC.FTC_On )
      Coil( #Sts.OP_CanMoveFreely )
   END_RUNG
   // the same network as SCL:
   "BTrk_Absence"(Item := "BTrk".A0301."B"["BTRK_A0301_Pos4_to_Pos5"], ENO => #_w1);
   "BTrk_Absence"(EN := #_w1, Item := "BTrk".A0301."B"["BTRK_A0301_Pos5_SpinLat1-2_Solleva"], ENO => #_w2);
   "BTrk_Absence"(EN := #_w2 OR (#Cin.P4.Fermi.Work AND #Cin.P5.Spintore_Lat.Spin_Lat1.Rest AND #Cin.P5.Spintore_Lat.Spin_Lat2.Rest AND #Cin.P5.Spintore_Lat.Sollevatori.Rest),
                  Item := "BTrk".A0301."B"["BTRK_A0301_Pos5.2_Long_PosAttesa"],
                  ENO => #_w3);
   "BTrk_Absence"(EN := #_w3, Item := "BTrk".A0301."B"["BTRK_A0302_SPINTORE"], ENO => #_w4);
   #Sts.OP_CanMoveFreely := #_w4;
   "BTrk_Absence"(EN := #Sts.OP_CanMoveFreely,
                  Item := "BTrk".A0301."B"["BTRK_A0302_SPINTORE_USCITA_TRASPORTO_A031"],
                  ENO => #_w5);
   "BTrk_Absence"(EN := #_w5, Item := "BTrk".A0301."B"["BTRK_A0302_SPINTORE_INGRESSO_BORDATRICE"], ENO => #_w6);
   #Sts.OP_CanMoveFreely := #_w6 AND NOT #IEC.FTC_On;
END_REGION

REGION Network 10: Ax - Comando Operazione Lavoro / Riposo (AUT)
   RUNG wire#powerrail
      Contact( #Cin.Manager.Control_ON )
      wire#w1
      Contact( #Cin.Manager.Rest )
      Coil( #Ctrl.Ax.OP_Rest_Aut )
   END_RUNG
   RUNG wire#w1
      Contact( #Cin.Manager.Work )
      Coil( #Ctrl.Ax.OP_Work_Aut )
   END_RUNG
   // the same network as SCL:
   #Ctrl.Ax.OP_Rest_Aut := #Cin.Manager.Control_ON AND #Cin.Manager.Rest;
   #Ctrl.Ax.OP_Work_Aut := #Cin.Manager.Control_ON AND #Cin.Manager.Work;
END_REGION

REGION Network 11: Ax - Comando Operazione Lavoro / Riposo (MAN)
   RUNG wire#powerrail
      P_Contact(operand := #DataIn.OP.Rest, bit := #AUX.OP_Rest_PB)
      Coil( #PE.OP_Rest_PB )
   END_RUNG
   RUNG wire#powerrail
      P_Contact(operand := #DataIn.OP.Work, bit := #AUX.OP_Work_PB)
      Coil( #PE.OP_Work_PB )
   END_RUNG
   RUNG wire#powerrail
      Contact( #AreaInterface.Man )
      I_Contact( #Cin.Manager.Control_ON )
      wire#w1
      Contact( #PE.OP_Rest_PB )
      wire#w2
      Contact( #DataIn.OP.Rest )
      I_Contact( #DataIn.OP.Work )
      Coil( #Ctrl.Ax.OP_Rest_Man )
   END_RUNG
   RUNG wire#w1
      Contact( #Ctrl.Ax.OP_Rest_Man )
   END_RUNG wire#w2
   RUNG wire#w1
      Contact( #PE.OP_Work_PB )
      wire#w3
      Contact( #DataIn.OP.Work )
      I_Contact( #DataIn.OP.Rest )
      Coil( #Ctrl.Ax.OP_Work_Man )
   END_RUNG
   RUNG wire#w1
      Contact( #Ctrl.Ax.OP_Work_Man )
   END_RUNG wire#w3
   // the same network as SCL:
   #_w1 := #DataIn.OP.Rest AND NOT #AUX.OP_Rest_PB;   // rising edge of #DataIn.OP.Rest
   #AUX.OP_Rest_PB := #DataIn.OP.Rest;
   #PE.OP_Rest_PB := #_w1;
   #_w2 := #DataIn.OP.Work AND NOT #AUX.OP_Work_PB;   // rising edge of #DataIn.OP.Work
   #AUX.OP_Work_PB := #DataIn.OP.Work;
   #PE.OP_Work_PB := #_w2;
   #_w3 := #AreaInterface.Man AND NOT #Cin.Manager.Control_ON;
   #Ctrl.Ax.OP_Rest_Man := #_w3 AND (#PE.OP_Rest_PB OR #Ctrl.Ax.OP_Rest_Man) AND #DataIn.OP.Rest AND NOT #DataIn.OP.Work;
   #Ctrl.Ax.OP_Work_Man := #_w3 AND (#PE.OP_Work_PB OR #Ctrl.Ax.OP_Work_Man) AND #DataIn.OP.Work AND NOT #DataIn.OP.Rest;
END_REGION

REGION Network 12: Ax - Cumulativo Operazione Lavoro / Riposo (ALL)
   RUNG wire#powerrail
      I_Contact( #Ctrl.Ax.OP_Rest_Man )
      I_Contact( #Ctrl.Ax.OP_Rest_Aut )
      Not()
      Coil( #Ctrl.Ax.OP_Rest )
   END_RUNG
   RUNG wire#powerrail
      I_Contact( #Ctrl.Ax.OP_Work_Man )
      I_Contact( #Ctrl.Ax.OP_Work_Aut )
      Not()
      Coil( #Ctrl.Ax.OP_Work )
   END_RUNG
   // the same network as SCL:
   #Ctrl.Ax.OP_Rest := NOT (NOT #Ctrl.Ax.OP_Rest_Man AND NOT #Ctrl.Ax.OP_Rest_Aut);
   #Ctrl.Ax.OP_Work := NOT (NOT #Ctrl.Ax.OP_Work_Man AND NOT #Ctrl.Ax.OP_Work_Aut);
END_REGION

REGION Network 13: Ax - Condizioni movimento Operazione a Lavoro / Riposo
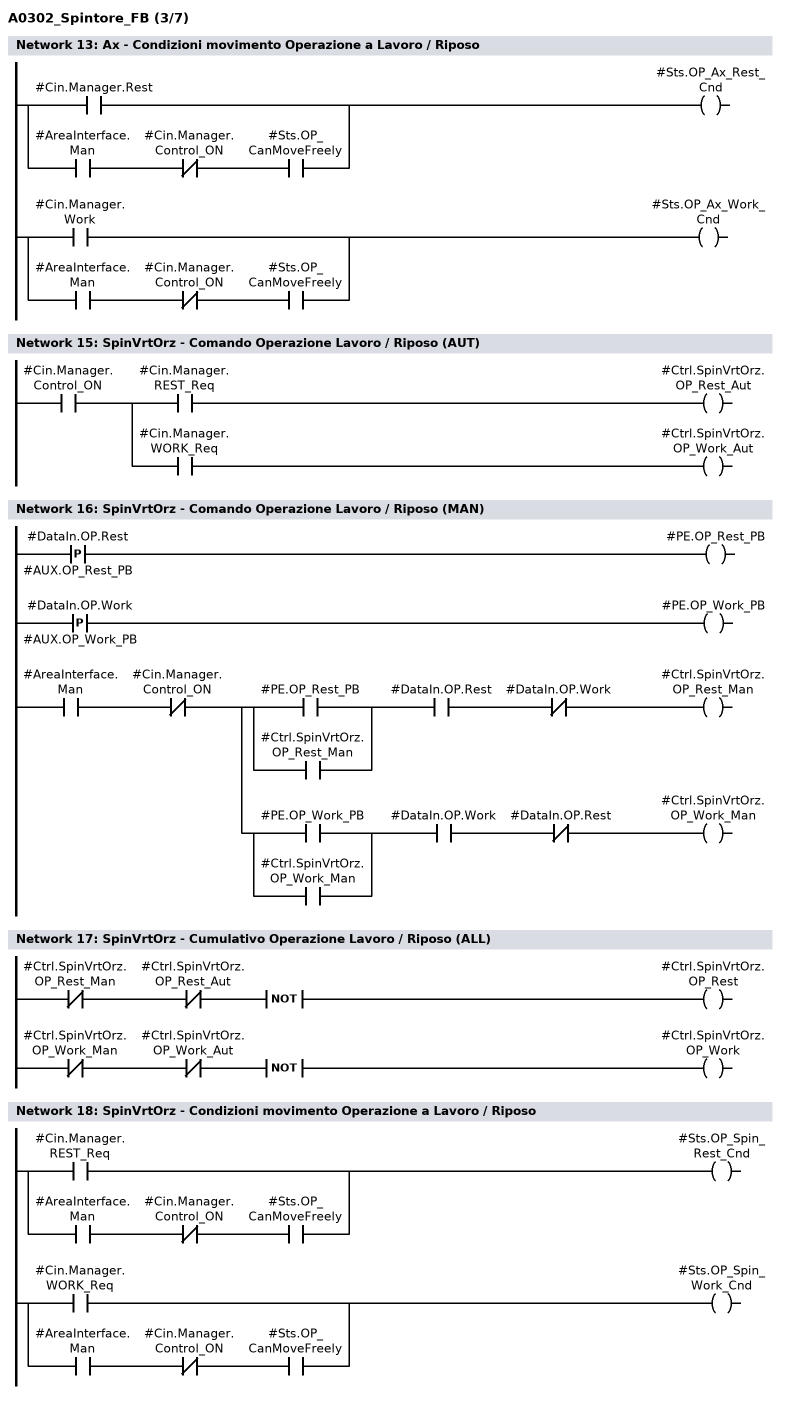
   RUNG wire#powerrail
      Contact( #Cin.Manager.Rest )
      wire#w1
      Coil( #Sts.OP_Ax_Rest_Cnd )
   END_RUNG
   RUNG wire#powerrail
      Contact( #AreaInterface.Man )
      I_Contact( #Cin.Manager.Control_ON )
      Contact( #Sts.OP_CanMoveFreely )
   END_RUNG wire#w1
   RUNG wire#powerrail
      Contact( #Cin.Manager.Work )
      wire#w2
      Coil( #Sts.OP_Ax_Work_Cnd )
   END_RUNG
   RUNG wire#powerrail
      Contact( #AreaInterface.Man )
      I_Contact( #Cin.Manager.Control_ON )
      Contact( #Sts.OP_CanMoveFreely )
   END_RUNG wire#w2
   // the same network as SCL:
   #Sts.OP_Ax_Rest_Cnd := #Cin.Manager.Rest OR (#AreaInterface.Man AND NOT #Cin.Manager.Control_ON AND #Sts.OP_CanMoveFreely);
   #Sts.OP_Ax_Work_Cnd := #Cin.Manager.Work OR (#AreaInterface.Man AND NOT #Cin.Manager.Control_ON AND #Sts.OP_CanMoveFreely);
END_REGION

REGION Network 15: SpinVrtOrz - Comando Operazione Lavoro / Riposo (AUT)
   RUNG wire#powerrail
      Contact( #Cin.Manager.Control_ON )
      wire#w1
      Contact( #Cin.Manager.REST_Req )
      Coil( #Ctrl.SpinVrtOrz.OP_Rest_Aut )
   END_RUNG
   RUNG wire#w1
      Contact( #Cin.Manager.WORK_Req )
      Coil( #Ctrl.SpinVrtOrz.OP_Work_Aut )
   END_RUNG
   // the same network as SCL:
   #Ctrl.SpinVrtOrz.OP_Rest_Aut := #Cin.Manager.Control_ON AND #Cin.Manager.REST_Req;
   #Ctrl.SpinVrtOrz.OP_Work_Aut := #Cin.Manager.Control_ON AND #Cin.Manager.WORK_Req;
END_REGION

REGION Network 16: SpinVrtOrz - Comando Operazione Lavoro / Riposo (MAN)
   RUNG wire#powerrail
      P_Contact(operand := #DataIn.OP.Rest, bit := #AUX.OP_Rest_PB)
      Coil( #PE.OP_Rest_PB )
   END_RUNG
   RUNG wire#powerrail
      P_Contact(operand := #DataIn.OP.Work, bit := #AUX.OP_Work_PB)
      Coil( #PE.OP_Work_PB )
   END_RUNG
   RUNG wire#powerrail
      Contact( #AreaInterface.Man )
      I_Contact( #Cin.Manager.Control_ON )
      wire#w1
      Contact( #PE.OP_Rest_PB )
      wire#w2
      Contact( #DataIn.OP.Rest )
      I_Contact( #DataIn.OP.Work )
      Coil( #Ctrl.SpinVrtOrz.OP_Rest_Man )
   END_RUNG
   RUNG wire#w1
      Contact( #Ctrl.SpinVrtOrz.OP_Rest_Man )
   END_RUNG wire#w2
   RUNG wire#w1
      Contact( #PE.OP_Work_PB )
      wire#w3
      Contact( #DataIn.OP.Work )
      I_Contact( #DataIn.OP.Rest )
      Coil( #Ctrl.SpinVrtOrz.OP_Work_Man )
   END_RUNG
   RUNG wire#w1
      Contact( #Ctrl.SpinVrtOrz.OP_Work_Man )
   END_RUNG wire#w3
   // the same network as SCL:
   #_w1 := #DataIn.OP.Rest AND NOT #AUX.OP_Rest_PB;   // rising edge of #DataIn.OP.Rest
   #AUX.OP_Rest_PB := #DataIn.OP.Rest;
   #PE.OP_Rest_PB := #_w1;
   #_w2 := #DataIn.OP.Work AND NOT #AUX.OP_Work_PB;   // rising edge of #DataIn.OP.Work
   #AUX.OP_Work_PB := #DataIn.OP.Work;
   #PE.OP_Work_PB := #_w2;
   #_w3 := #AreaInterface.Man AND NOT #Cin.Manager.Control_ON;
   #Ctrl.SpinVrtOrz.OP_Rest_Man := #_w3 AND (#PE.OP_Rest_PB OR #Ctrl.SpinVrtOrz.OP_Rest_Man) AND #DataIn.OP.Rest AND NOT #DataIn.OP.Work;
   #Ctrl.SpinVrtOrz.OP_Work_Man := #_w3 AND (#PE.OP_Work_PB OR #Ctrl.SpinVrtOrz.OP_Work_Man) AND #DataIn.OP.Work AND NOT #DataIn.OP.Rest;
END_REGION

REGION Network 17: SpinVrtOrz - Cumulativo Operazione Lavoro / Riposo (ALL)
   RUNG wire#powerrail
      I_Contact( #Ctrl.SpinVrtOrz.OP_Rest_Man )
      I_Contact( #Ctrl.SpinVrtOrz.OP_Rest_Aut )
      Not()
      Coil( #Ctrl.SpinVrtOrz.OP_Rest )
   END_RUNG
   RUNG wire#powerrail
      I_Contact( #Ctrl.SpinVrtOrz.OP_Work_Man )
      I_Contact( #Ctrl.SpinVrtOrz.OP_Work_Aut )
      Not()
      Coil( #Ctrl.SpinVrtOrz.OP_Work )
   END_RUNG
   // the same network as SCL:
   #Ctrl.SpinVrtOrz.OP_Rest := NOT (NOT #Ctrl.SpinVrtOrz.OP_Rest_Man AND NOT #Ctrl.SpinVrtOrz.OP_Rest_Aut);
   #Ctrl.SpinVrtOrz.OP_Work := NOT (NOT #Ctrl.SpinVrtOrz.OP_Work_Man AND NOT #Ctrl.SpinVrtOrz.OP_Work_Aut);
END_REGION

REGION Network 18: SpinVrtOrz - Condizioni movimento Operazione a Lavoro / Riposo
   RUNG wire#powerrail
      Contact( #Cin.Manager.REST_Req )
      wire#w1
      Coil( #Sts.OP_Spin_Rest_Cnd )
   END_RUNG
   RUNG wire#powerrail
      Contact( #AreaInterface.Man )
      I_Contact( #Cin.Manager.Control_ON )
      Contact( #Sts.OP_CanMoveFreely )
   END_RUNG wire#w1
   RUNG wire#powerrail
      Contact( #Cin.Manager.WORK_Req )
      wire#w2
      Coil( #Sts.OP_Spin_Work_Cnd )
   END_RUNG
   RUNG wire#powerrail
      Contact( #AreaInterface.Man )
      I_Contact( #Cin.Manager.Control_ON )
      Contact( #Sts.OP_CanMoveFreely )
   END_RUNG wire#w2
   // the same network as SCL:
   #Sts.OP_Spin_Rest_Cnd := #Cin.Manager.REST_Req OR (#AreaInterface.Man AND NOT #Cin.Manager.Control_ON AND #Sts.OP_CanMoveFreely);
   #Sts.OP_Spin_Work_Cnd := #Cin.Manager.WORK_Req OR (#AreaInterface.Man AND NOT #Cin.Manager.Control_ON AND #Sts.OP_CanMoveFreely);
END_REGION

REGION Network 20 (SCL): Verticale + Orizzontale + Ax - Cin Manager (Esecuzione sequenza comandi)
   #Ax.CIn.Manager.Control_ON:= #Cin.Manager.Control_ON;
   #Orz.Cin.Manager.Control_ON := #Vrt.Cin.Manager.Control_ON := #Cin.Manager.Control_ON;


   #Vrt.Cin.Manager.Rest := FALSE;
   #Vrt.Cin.Manager.Work := FALSE;
   #Orz.Cin.Manager.Rest := FALSE;
   #Orz.Cin.Manager.Work := FALSE;
   #Ax.CIn.Manager.MoveToPos := FALSE;


   // Operazione riposo del cilindro verticale ed orizzontale sullo spintore
   IF (#Ctrl.SpinVrtOrz.OP_Rest OR #Cin.Manager.REST_Req) AND #Sts.OP_Spin_Rest_Cnd THEN

       #Orz.Cin.Manager.Rest := #Orz.COut.Rest := TRUE;
       #Vrt.Cin.Manager.Rest := #Vrt.COut.Rest := #Orz.COut.Rest;

       // Operazione lavoro del cilindro verticale ed orizzontale sullo spintore   
   ELSIF (#Ctrl.SpinVrtOrz.OP_Work OR #Cin.Manager.WORK_Req) AND #Sts.OP_Spin_Work_Cnd THEN

       #Vrt.Cin.Manager.Work := #Vrt.COut.Work := TRUE;
       #Orz.Cin.Manager.Work := #Vrt.Cin.Manager.Work;

   END_IF;

   // Operazione arresto dell' asse spintore quando i 2 ciclindri sono in riposo
   IF #Ctrl.Ax.OP_Rest AND #Sts.OP_Ax_Rest_Cnd THEN
       #Ax.CIn.Manager.Pos := #Data.Ax_Pos.PosAttesa;
       #Ax.CIn.Manager.Vel := #Par_Ax_Auto.Aut_Vel;
       #Ax.CIn.Manager.Acc := #Par_Ax_Auto.Aut_Acc;
       #Ax.CIn.Manager.Dec := #Par_Ax_Auto.Aut_Dec;
       #Ax.CIn.Manager.MoveToPos := TRUE;

       // Se raggiungo la pos.attesa spengo il comando
   ELSIF #Ctrl.Ax.OP_Rest AND #Sts.OP_Ax_Rest_Cnd AND #COut.Ax_Sts.PosAttesa_Reached THEN
       #Ax.CIn.Manager.MoveToPos := #Ax.CIn.Manager.Control_ON := FALSE;

   END_IF;

   // Operazione lavoro dell' asse spintore quando i 2 ciclindri sono in lavoro
   IF #Ctrl.Ax.OP_Work AND #Sts.OP_Ax_Work_Cnd AND #Vrt.COut.Work AND #Orz.COut.Work
        AND NOT #Alarm.Orz_AnalSens_Compressed THEN
       #Ax.CIn.Manager.Pos := #Data.Ax_Pos.PosFineSpinta;
       #Ax.CIn.Manager.Vel := #Par_Ax_Auto.Aut_Vel;
       #Ax.CIn.Manager.Acc := #Par_Ax_Auto.Aut_Acc;
       #Ax.CIn.Manager.Dec := #Par_Ax_Auto.Aut_Dec;
       #Ax.CIn.Manager.MoveToPos := TRUE;

      // Se raggiungo la pos. o il sensore viene compresso disabilito la spinta 
   ELSIF (#Ctrl.Ax.OP_Work AND #Sts.OP_Ax_Work_Cnd) AND #COut.Ax_Sts.PosFineSpinta_Reached THEN
       #Ax.CIn.Manager.MoveToPos := FALSE;

   ELSIF (#Ctrl.Ax.OP_Work AND #Sts.OP_Ax_Work_Cnd) AND #Alarm.Orz_AnalSens_Compressed THEN
       #Ax.CIn.Manager.MoveToPos := FALSE;

   END_IF;
END_REGION

REGION Network 21 (SCL): Verticale + Orizzontale + Ax - CIn Abilitazioni Stop Manager
   #Vrt.Cin.Manager.EnableStopDoorOpeningReq := #Orz.Cin.Manager.EnableStopDoorOpeningReq
   := #Ax.CIn.Manager.EnableStopDoorOpeningReq := #Cin.Manager.EnableStopDoorOpeningReq;

   #Vrt.Cin.Manager.EnableStopInPhase := #Orz.Cin.Manager.EnableStopInPhase
   := #Ax.CIn.Manager.EnableStopInPhase := #Cin.Manager.EnableStopInPhase;

   #Vrt.Cin.Manager.EnableStopProgrammed := #Orz.Cin.Manager.EnableStopProgrammed
   := #Ax.CIn.Manager.EnableStopProgrammed := #Cin.Manager.EnableStopProgrammed;
END_REGION

REGION Network 22: <+>
END_REGION

REGION Network 23: Warning manacanza condizioni esecuzione Operazione RIPOSO / LAVORO
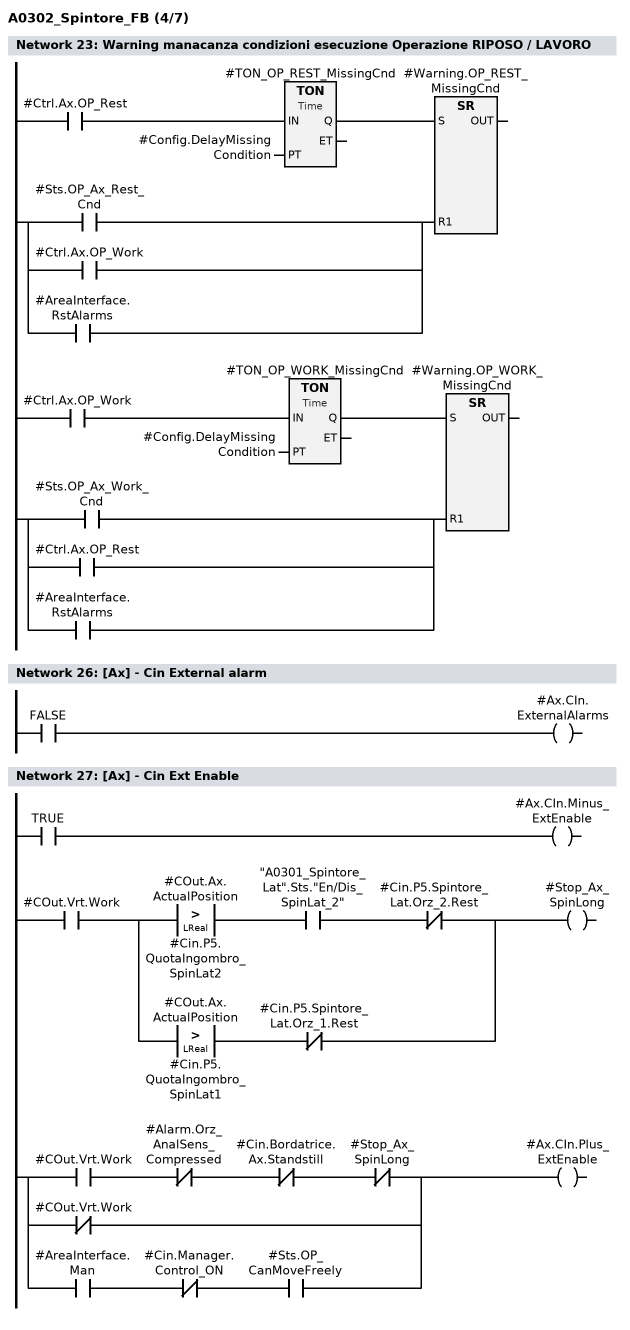
   RUNG wire#powerrail
      Contact( #Ctrl.Ax.OP_Rest )
      { S7_Templates := "time_type := Time" } #TON_OP_REST_MissingCnd.TON(pt := #Config.DelayMissingCondition, et =>)
      S_SR(operand := #Warning.OP_REST_MissingCnd, r1 := wire#w1)
   END_RUNG
   RUNG wire#powerrail
      Contact( #Sts.OP_Ax_Rest_Cnd )
   END_RUNG wire#w1
   RUNG wire#powerrail
      Contact( #Ctrl.Ax.OP_Work )
   END_RUNG wire#w1
   RUNG wire#powerrail
      Contact( #AreaInterface.RstAlarms )
   END_RUNG wire#w1
   RUNG wire#powerrail
      Contact( #Ctrl.Ax.OP_Work )
      { S7_Templates := "time_type := Time" } #TON_OP_WORK_MissingCnd.TON(pt := #Config.DelayMissingCondition, et =>)
      S_SR(operand := #Warning.OP_WORK_MissingCnd, r1 := wire#w2)
   END_RUNG
   RUNG wire#powerrail
      Contact( #Sts.OP_Ax_Work_Cnd )
   END_RUNG wire#w2
   RUNG wire#powerrail
      Contact( #Ctrl.Ax.OP_Rest )
   END_RUNG wire#w2
   RUNG wire#powerrail
      Contact( #AreaInterface.RstAlarms )
   END_RUNG wire#w2
   // the same network as SCL:
   #TON_OP_REST_MissingCnd(IN := #Ctrl.Ax.OP_Rest, PT := #Config.DelayMissingCondition);   // TON
   IF #TON_OP_REST_MissingCnd.Q THEN
       #Warning.OP_REST_MissingCnd := TRUE;   // SR flip-flop
   END_IF;
   IF #Sts.OP_Ax_Rest_Cnd OR #Ctrl.Ax.OP_Work OR #AreaInterface.RstAlarms THEN
       #Warning.OP_REST_MissingCnd := FALSE;
   END_IF;
   #TON_OP_WORK_MissingCnd(IN := #Ctrl.Ax.OP_Work, PT := #Config.DelayMissingCondition);   // TON
   IF #TON_OP_WORK_MissingCnd.Q THEN
       #Warning.OP_WORK_MissingCnd := TRUE;   // SR flip-flop
   END_IF;
   IF #Sts.OP_Ax_Work_Cnd OR #Ctrl.Ax.OP_Rest OR #AreaInterface.RstAlarms THEN
       #Warning.OP_WORK_MissingCnd := FALSE;
   END_IF;
END_REGION

REGION Network 25 (SCL): << RIFERIMENTI [Spintore Ax] - Positioning Manager >>
   // ******************************************************************************************
   REGION // TRASFERIMENTO DELLE RAMPE

       // Rampe in Automatico o Semi-Automatico
       IF #AreaInterface.Aut AND NOT #Cin.SemiAut_Pb THEN
           #Ax.CIn.Manager.Acc := #Par_Ax_Auto.Aut_Acc;
           #Ax.CIn.Manager.Dec := #Par_Ax_Auto.Aut_Dec;
       ELSIF #Cin.SemiAut_Pb THEN
           #Ax.CIn.Manager.Acc := #Par_Ax_Auto.Aut_Acc;
           #Ax.CIn.Manager.Dec := #Par_Ax_Auto.Aut_Dec;
       END_IF;

       // Rampe in Manuale
       IF #AreaInterface.Man AND NOT #Cin.SemiAut_Pb THEN
           #Ax.CIn.Manager.Acc := #Par_Ax_Manu.Man_Acc;
           #Ax.CIn.Manager.Dec := #Par_Ax_Manu.Man_Dec;
       END_IF;
   END_REGION

   // ******************************************************************************************
   REGION // // CALCOLO DELLA VELOCITA' TRASFERITA AL DRIVE IN BASE AL CALCOLO DEL CICLINDRO COMPENSATORE
       (*
   #Sts.ResiduoCilindro := #CorsaCilindro - #Sts.PosCilindro;

   #Sts.spazio_frenata := ((#Ctrl.Vel / 60.0) ** 2.0) /(2.0 * #Ctrl.Dec);

   #SpazioSafe := #Sts.spazio_frenata + #Par.CylComp_SafeResidual;

   #Ctrl.StopSicurezza := (#Sts.ResiduoCilindro - #SpazioSafe) < 0.0;

   // bisogna calcolare la decelerazione massima per rispettare frenata
   // 
   #Sts.DecMassima := ((#Ctrl.Vel / 60.0) ** 2.0) / (2 * (#Sts.ResiduoCilindro - #Par.CylComp_SafeResidual));
   *)

       // Velocità asse in base alla velocità della chiudi bordi..
       #Ctrl.Ax.Vel := #Cin.Bordatrice.TargetVel * #Cin.Bordatrice.Perc_Vel / 100.0;

       // Limite decellerazione dell'asse
       #DecMax := (#Ax.Config.Ax.MaxDec_S120_P2573 / 1000.0);

   (*// Spazio di frenata da raggiungere
   // 
   #SpazioSafe := #CorsaCilindroCompensatore - #Par.Spintore.Compensatore_SpazioResiduoExtra;
   *)

       // Nuovo valore di velocità per limitare e rispettare spazio di arresto con massima decelerazione possibile
       // 
       #Ctrl.Ax.VelMax := LREAL_TO_REAL(IN:= (60.0 * (SQRT(2.0 * #DecMax * #Orz_SpazioSafe))));

       // Limitazione della velocità per rispettare lo spazio di frenata   
       #Ctrl.Ax.Vel := MIN_REAL(IN1 := #Ctrl.Ax.Vel, IN2 := #Ctrl.Ax.VelMax);

   END_REGION ;

   // *****************************************************************************************
   REGION // CALCOLO DELLA VELOCITA' E TRASFERIMENTO IN BASE ALLO STATO IMPIANTO
       //
       IF NOT #Ax.CIn.Manager.Control_ON THEN
           // CALCOLO VELOCITA' IN BASE ALL'OVERIDE
           IF #Ax.AreaInterface.Aut THEN
               #Ax.CIn.Manager.Vel := #Ctrl.Ax.Vel;
           ELSIF #Cin.SemiAut_Pb THEN
               #Ax.CIn.Manager.Vel := (#Par_Ax_Auto.SemiAut_Vel * #Ctrl.Ax.Vel);
           END_IF;
       END_IF;
   END_REGION ;
END_REGION

REGION Network 26: [Ax] - Cin External alarm
   RUNG wire#powerrail
      Contact( FALSE )
      Coil( #Ax.CIn.ExternalAlarms )
   END_RUNG
   // the same network as SCL:
   #Ax.CIn.ExternalAlarms := FALSE;
END_REGION

REGION Network 27: [Ax] - Cin Ext Enable
   RUNG wire#powerrail
      Contact( TRUE )
      Coil( #Ax.CIn.Minus_ExtEnable )
   END_RUNG
   RUNG wire#powerrail
      Contact( #COut.Vrt.Work )
      wire#w1
      { S7_Templates := "SrcType := LReal" } GT_Contact(in1 := #COut.Ax.ActualPosition, in2 := #Cin.P5.QuotaIngombro_SpinLat2)
      Contact( "A0301_Spintore_Lat".Sts."En/Dis_SpinLat_2" )
      I_Contact( #Cin.P5.Spintore_Lat.Orz_2.Rest )
      wire#w2
      Coil( #Stop_Ax_SpinLong )
   END_RUNG
   RUNG wire#w1
      { S7_Templates := "SrcType := LReal" } GT_Contact(in1 := #COut.Ax.ActualPosition, in2 := #Cin.P5.QuotaIngombro_SpinLat1)
      I_Contact( #Cin.P5.Spintore_Lat.Orz_1.Rest )
   END_RUNG wire#w2
   RUNG wire#powerrail
      Contact( #COut.Vrt.Work )
      I_Contact( #Alarm.Orz_AnalSens_Compressed )
      I_Contact( #Cin.Bordatrice.Ax.Standstill )
      I_Contact( #Stop_Ax_SpinLong )
      wire#w3
      Coil( #Ax.CIn.Plus_ExtEnable )
   END_RUNG
   RUNG wire#powerrail
      I_Contact( #COut.Vrt.Work )
   END_RUNG wire#w3
   RUNG wire#powerrail
      Contact( #AreaInterface.Man )
      I_Contact( #Cin.Manager.Control_ON )
      Contact( #Sts.OP_CanMoveFreely )
   END_RUNG wire#w3
   // the same network as SCL:
   #Ax.CIn.Minus_ExtEnable := TRUE;
   #Stop_Ax_SpinLong := #COut.Vrt.Work AND (((#COut.Ax.ActualPosition > #Cin.P5.QuotaIngombro_SpinLat2) AND "A0301_Spintore_Lat".Sts."En/Dis_SpinLat_2" AND NOT #Cin.P5.Spintore_Lat.Orz_2.Rest) OR ((#COut.Ax.ActualPosition > #Cin.P5.QuotaIngombro_SpinLat1) AND NOT #Cin.P5.Spintore_Lat.Orz_1.Rest));
   #Ax.CIn.Plus_ExtEnable := (#COut.Vrt.Work AND NOT #Alarm.Orz_AnalSens_Compressed AND NOT #Cin.Bordatrice.Ax.Standstill AND NOT #Stop_Ax_SpinLong) OR NOT #COut.Vrt.Work OR (#AreaInterface.Man AND NOT #Cin.Manager.Control_ON AND #Sts.OP_CanMoveFreely);
END_REGION

REGION Network 28: [Ax] HMI preset position
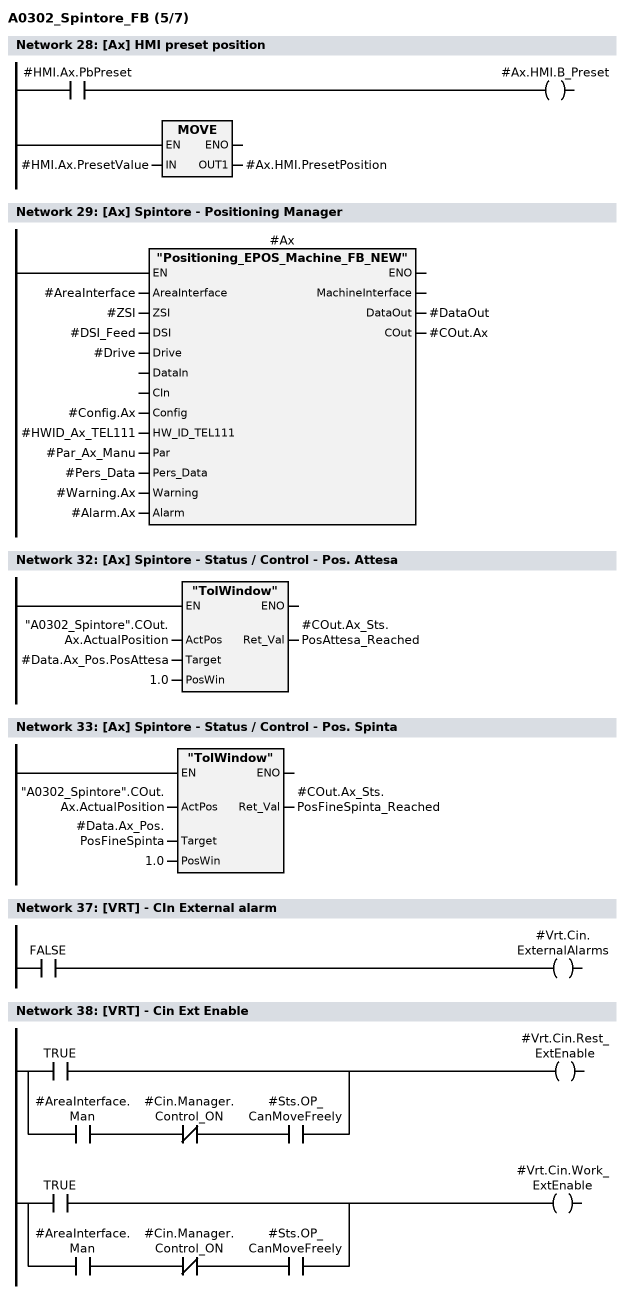
   RUNG wire#powerrail
      Contact( #HMI.Ax.PbPreset )
      Coil( #Ax.HMI.B_Preset )
   END_RUNG
   RUNG wire#powerrail
      Move(in := #HMI.Ax.PresetValue, out1 => #Ax.HMI.PresetPosition)
   END_RUNG
   // the same network as SCL:
   #Ax.HMI.B_Preset := #HMI.Ax.PbPreset;
   #Ax.HMI.PresetPosition := #HMI.Ax.PresetValue;
END_REGION

REGION Network 29: [Ax] Spintore - Positioning Manager
   RUNG wire#powerrail
      #Ax(AreaInterface := #AreaInterface, ZSI := #ZSI, DSI := #DSI_Feed, Drive := #Drive, DataIn :=, CIn :=, Config := #Config.Ax, HW_ID_TEL111 := #HWID_Ax_TEL111, Par := #Par_Ax_Manu, Pers_Data := #Pers_Data, Warning := #Warning.Ax, Alarm := #Alarm.Ax, MachineInterface =>, DataOut => #DataOut, COut => #COut.Ax)
   END_RUNG
   // the same network as SCL:
   #Ax(AreaInterface := #AreaInterface,   // "Positioning_EPOS_Machine_FB_NEW"
       ZSI := #ZSI,
       DSI := #DSI_Feed,
       Drive := #Drive,
       Config := #Config.Ax,
       HW_ID_TEL111 := #HWID_Ax_TEL111,
       Par := #Par_Ax_Manu,
       Pers_Data := #Pers_Data,
       Warning := #Warning.Ax,
       Alarm := #Alarm.Ax,
       DataOut => #DataOut,
       COut => #COut.Ax);
END_REGION

REGION Network 30: <+>
END_REGION

REGION Network 31: <<< CONTROLLO REQ da TRAKING E CAMBIO POS. >>>
END_REGION

REGION Network 32: [Ax] Spintore - Status / Control - Pos. Attesa
   RUNG wire#powerrail
      "TolWindow"(ActPos := "A0302_Spintore".COut.Ax.ActualPosition, Target := #Data.Ax_Pos.PosAttesa, PosWin := 1.0, Ret_Val => #COut.Ax_Sts.PosAttesa_Reached)
   END_RUNG
   // the same network as SCL:
   #COut.Ax_Sts.PosAttesa_Reached := "TolWindow"(ActPos := "A0302_Spintore".COut.Ax.ActualPosition,
                           Target := #Data.Ax_Pos.PosAttesa,
                           PosWin := 1.0);
END_REGION

REGION Network 33: [Ax] Spintore - Status / Control - Pos. Spinta
   RUNG wire#powerrail
      "TolWindow"(ActPos := "A0302_Spintore".COut.Ax.ActualPosition, Target := #Data.Ax_Pos.PosFineSpinta, PosWin := 1.0, Ret_Val => #COut.Ax_Sts.PosFineSpinta_Reached)
   END_RUNG
   // the same network as SCL:
   #COut.Ax_Sts.PosFineSpinta_Reached := "TolWindow"(ActPos := "A0302_Spintore".COut.Ax.ActualPosition,
                           Target := #Data.Ax_Pos.PosFineSpinta,
                           PosWin := 1.0);
END_REGION

REGION Network 34: <+>
END_REGION

REGION Network 36: <<< SPINTORE LONGITUDINALE - VRT >>>
END_REGION

REGION Network 37: [VRT] - CIn External alarm
   RUNG wire#powerrail
      Contact( FALSE )
      Coil( #Vrt.Cin.ExternalAlarms )
   END_RUNG
   // the same network as SCL:
   #Vrt.Cin.ExternalAlarms := FALSE;
END_REGION

REGION Network 38: [VRT] - Cin Ext Enable
   RUNG wire#powerrail
      Contact( TRUE )
      wire#w1
      Coil( #Vrt.Cin.Rest_ExtEnable )
   END_RUNG
   RUNG wire#powerrail
      Contact( #AreaInterface.Man )
      I_Contact( #Cin.Manager.Control_ON )
      Contact( #Sts.OP_CanMoveFreely )
   END_RUNG wire#w1
   RUNG wire#powerrail
      Contact( TRUE )
      wire#w2
      Coil( #Vrt.Cin.Work_ExtEnable )
   END_RUNG
   RUNG wire#powerrail
      Contact( #AreaInterface.Man )
      I_Contact( #Cin.Manager.Control_ON )
      Contact( #Sts.OP_CanMoveFreely )
   END_RUNG wire#w2
   // the same network as SCL:
   #Vrt.Cin.Rest_ExtEnable := TRUE OR (#AreaInterface.Man AND NOT #Cin.Manager.Control_ON AND #Sts.OP_CanMoveFreely);
   #Vrt.Cin.Work_ExtEnable := TRUE OR (#AreaInterface.Man AND NOT #Cin.Manager.Control_ON AND #Sts.OP_CanMoveFreely);
END_REGION

REGION Network 39: [VRT] - Valve Manager
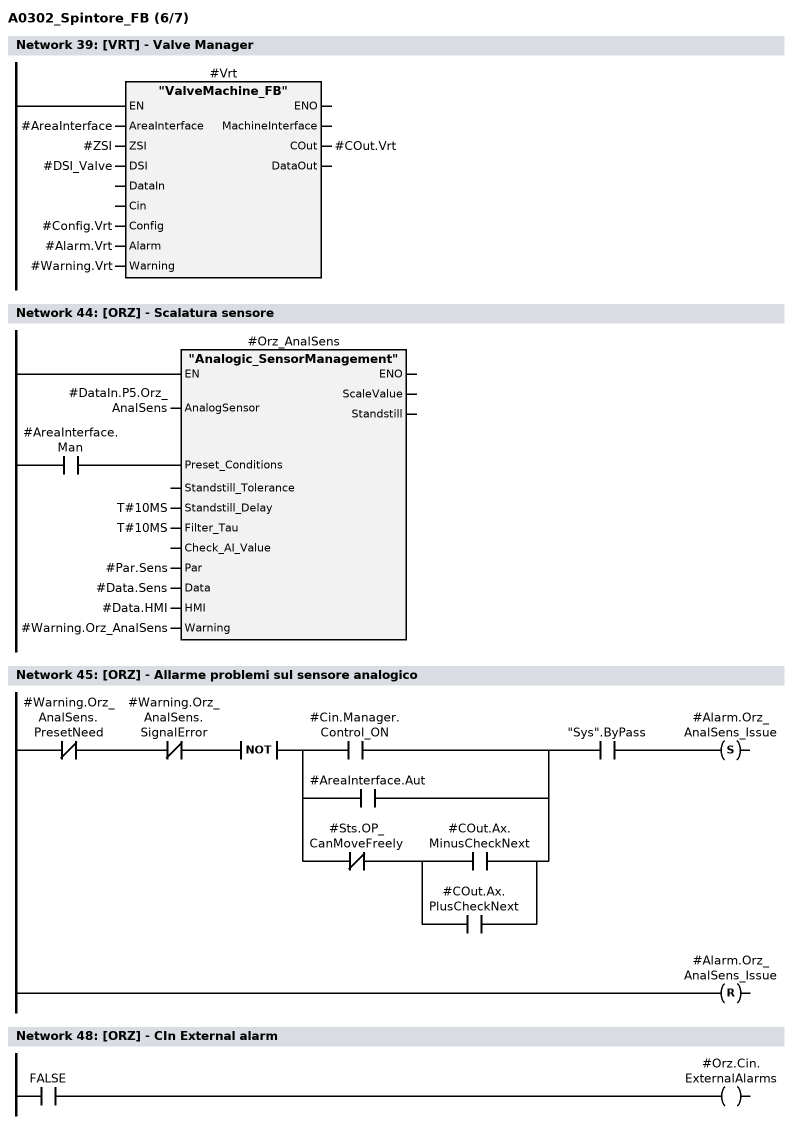
   RUNG wire#powerrail
      #Vrt(AreaInterface := #AreaInterface, ZSI := #ZSI, DSI := #DSI_Valve, DataIn :=, Cin :=, Config := #Config.Vrt, Alarm := #Alarm.Vrt, Warning := #Warning.Vrt, MachineInterface =>, COut => #COut.Vrt, DataOut =>)
   END_RUNG
   // the same network as SCL:
   #Vrt(AreaInterface := #AreaInterface,   // "ValveMachine_FB"
        ZSI := #ZSI,
        DSI := #DSI_Valve,
        Config := #Config.Vrt,
        Alarm := #Alarm.Vrt,
        Warning := #Warning.Vrt,
        COut => #COut.Vrt);
END_REGION

REGION Network 41: <<< SPINTORE LONGITUDINALE - ORZ >>>
END_REGION

REGION Network 42: <+>
END_REGION

REGION Network 43: << GESTIONE SPINTORE ORIZ ANALOGIC SENSOR >>
END_REGION

REGION Network 44: [ORZ] - Scalatura sensore
   RUNG wire#powerrail
      #Orz_AnalSens(Preset_Conditions := wire#w1, AnalogSensor := #DataIn.P5.Orz_AnalSens, Standstill_Tolerance :=, Standstill_Delay := T#10MS, Filter_Tau := T#10MS, Check_AI_Value :=, Par := #Par.Sens, Data := #Data.Sens, HMI := #Data.HMI, Warning := #Warning.Orz_AnalSens, ScaleValue =>, Standstill =>)
   END_RUNG
   RUNG wire#powerrail
      Contact( #AreaInterface.Man )
   END_RUNG wire#w1
   // the same network as SCL:
   #Orz_AnalSens(AnalogSensor := #DataIn.P5.Orz_AnalSens,   // "Analogic_SensorManagement"
                 Preset_Conditions := #AreaInterface.Man,
                 Standstill_Delay := T#10MS,
                 Filter_Tau := T#10MS,
                 Par := #Par.Sens,
                 Data := #Data.Sens,
                 HMI := #Data.HMI,
                 Warning := #Warning.Orz_AnalSens);
END_REGION

REGION Network 45: [ORZ] - Allarme problemi sul sensore analogico
   RUNG wire#powerrail
      I_Contact( #Warning.Orz_AnalSens.PresetNeed )
      I_Contact( #Warning.Orz_AnalSens.SignalError )
      Not()
      wire#w1
      Contact( #Cin.Manager.Control_ON )
      wire#w2
      Contact( "Sys".ByPass )
      S_Coil( #Alarm.Orz_AnalSens_Issue )
   END_RUNG
   RUNG wire#w1
      Contact( #AreaInterface.Aut )
   END_RUNG wire#w2
   RUNG wire#w1
      I_Contact( #Sts.OP_CanMoveFreely )
      wire#w3
      Contact( #COut.Ax.MinusCheckNext )
   END_RUNG wire#w2
   RUNG wire#w3
      Contact( #COut.Ax.PlusCheckNext )
   END_RUNG wire#w2
   RUNG wire#powerrail
      R_Coil( #Alarm.Orz_AnalSens_Issue )
   END_RUNG
   // the same network as SCL:
   IF NOT (NOT #Warning.Orz_AnalSens.PresetNeed AND NOT #Warning.Orz_AnalSens.SignalError) AND (#Cin.Manager.Control_ON OR #AreaInterface.Aut OR (NOT #Sts.OP_CanMoveFreely AND (#COut.Ax.MinusCheckNext OR #COut.Ax.PlusCheckNext))) AND "Sys".ByPass THEN
       #Alarm.Orz_AnalSens_Issue := TRUE;
   END_IF;
   #Alarm.Orz_AnalSens_Issue := FALSE;
END_REGION

REGION Network 46 (SCL): [ORZ] - Calcolo range lavoro sensore
       // ********************************************************************************************************************************************
       // Calcolo lo spazio di sicurezza se ho eseguito il preset del sensore
       // Spazio di frenata da raggiungere

       IF #Par.Sens.Enable THEN
           IF #Data.Sens.OffsetValid THEN
               #Orz_SpazioSafe := #Par.Sens.RangeHigh - #Par_Mach.Tol_Work  ;
           END_IF;

           // Controllo finestra di lavoro del sensore, dato il valore di lavoro sicuro,se è inferiore sino in compressione sul pezzo.  
           IF  #Data.Sens.OffsetValid AND #Orz_SpazioSafe <> 0 AND 
               (#Orz_AnalSens.ScaleValue < (#Par.Sens.RangeHigh - #Orz_SpazioSafe)) THEN
               #Alarm.Orz_AnalSens_Compressed := 1;
           ELSE
               #Alarm.Orz_AnalSens_Compressed := 0;
           END_IF;
       END_IF;
END_REGION

REGION Network 47: <+>
END_REGION

REGION Network 48: [ORZ] - CIn External alarm
   RUNG wire#powerrail
      Contact( FALSE )
      Coil( #Orz.Cin.ExternalAlarms )
   END_RUNG
   // the same network as SCL:
   #Orz.Cin.ExternalAlarms := FALSE;
END_REGION

REGION Network 49: [ORZ] - Cin Ext Enable
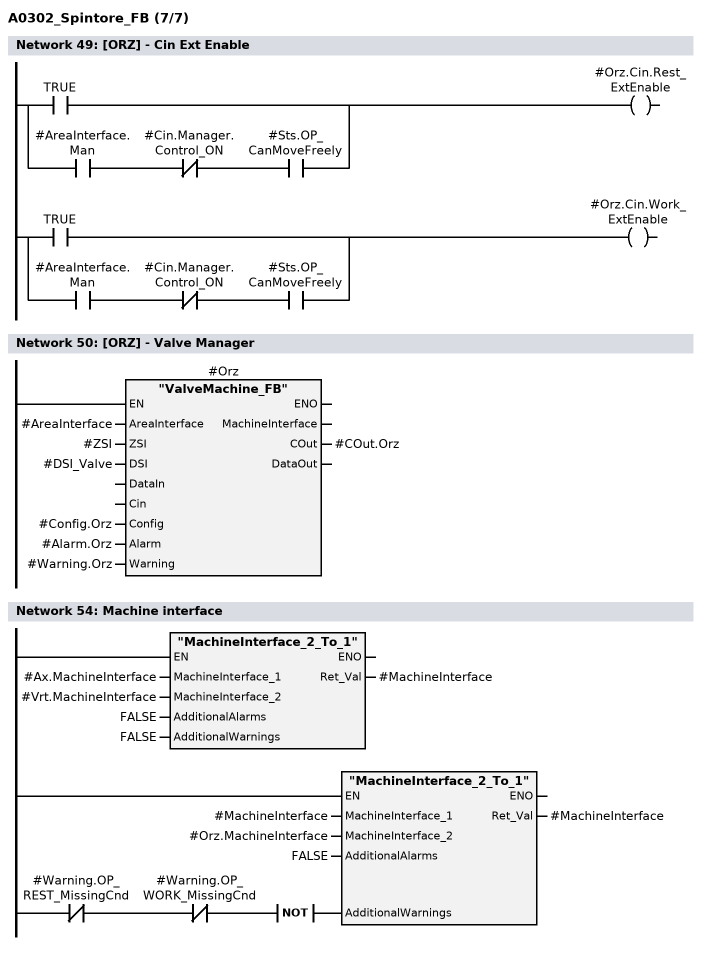
   RUNG wire#powerrail
      Contact( TRUE )
      wire#w1
      Coil( #Orz.Cin.Rest_ExtEnable )
   END_RUNG
   RUNG wire#powerrail
      Contact( #AreaInterface.Man )
      I_Contact( #Cin.Manager.Control_ON )
      Contact( #Sts.OP_CanMoveFreely )
   END_RUNG wire#w1
   RUNG wire#powerrail
      Contact( TRUE )
      wire#w2
      Coil( #Orz.Cin.Work_ExtEnable )
   END_RUNG
   RUNG wire#powerrail
      Contact( #AreaInterface.Man )
      I_Contact( #Cin.Manager.Control_ON )
      Contact( #Sts.OP_CanMoveFreely )
   END_RUNG wire#w2
   // the same network as SCL:
   #Orz.Cin.Rest_ExtEnable := TRUE OR (#AreaInterface.Man AND NOT #Cin.Manager.Control_ON AND #Sts.OP_CanMoveFreely);
   #Orz.Cin.Work_ExtEnable := TRUE OR (#AreaInterface.Man AND NOT #Cin.Manager.Control_ON AND #Sts.OP_CanMoveFreely);
END_REGION

REGION Network 50: [ORZ] - Valve Manager
   RUNG wire#powerrail
      #Orz(AreaInterface := #AreaInterface, ZSI := #ZSI, DSI := #DSI_Valve, DataIn :=, Cin :=, Config := #Config.Orz, Alarm := #Alarm.Orz, Warning := #Warning.Orz, MachineInterface =>, COut => #COut.Orz, DataOut =>)
   END_RUNG
   // the same network as SCL:
   #Orz(AreaInterface := #AreaInterface,   // "ValveMachine_FB"
        ZSI := #ZSI,
        DSI := #DSI_Valve,
        Config := #Config.Orz,
        Alarm := #Alarm.Orz,
        Warning := #Warning.Orz,
        COut => #COut.Orz);
END_REGION

REGION Network 51: <+>
END_REGION

REGION Network 52 (SCL): Stazione COut
   // VALVOLE SPINTORE
   #COut.Spintore.Standstill := #Vrt.COut.Standstill AND #Orz.COut.Standstill;
   #COut.Spintore.Rest_CheckNext := #Ctrl.Ax.OP_Rest AND #Ctrl.SpinVrtOrz.OP_Rest;
   #COut.Spintore.Work_CheckNext := #Ctrl.Ax.OP_Work AND #Ctrl.SpinVrtOrz.OP_Work ;
   #COut.Spintore.Rest := #Vrt.COut.Rest AND #Orz.COut.Rest;
   #COut.Spintore.Work := #Vrt.COut.Work AND #Orz.COut.Work;

   // SPINTORE LONGITUDINALE
   #COut.Ax := #Ax.COut;
   #COut.Vrt := #Vrt.COut;
   #COut.Orz := #Orz.COut;
END_REGION

REGION Network 53: <<< MACHINE STATUS >>>
END_REGION

REGION Network 54: Machine interface
   RUNG wire#powerrail
      "MachineInterface_2_To_1"(MachineInterface_1 := #Ax.MachineInterface, MachineInterface_2 := #Vrt.MachineInterface, AdditionalAlarms := FALSE, AdditionalWarnings := FALSE, Ret_Val => #MachineInterface)
   END_RUNG
   RUNG wire#powerrail
      "MachineInterface_2_To_1"(AdditionalWarnings := wire#w1, MachineInterface_1 := #MachineInterface, MachineInterface_2 := #Orz.MachineInterface, AdditionalAlarms := FALSE, Ret_Val => #MachineInterface)
   END_RUNG
   RUNG wire#powerrail
      I_Contact( #Warning.OP_REST_MissingCnd )
      I_Contact( #Warning.OP_WORK_MissingCnd )
      Not()
   END_RUNG wire#w1
   // the same network as SCL:
   #MachineInterface := "MachineInterface_2_To_1"(MachineInterface_1 := #Ax.MachineInterface,
                           MachineInterface_2 := #Vrt.MachineInterface,
                           AdditionalAlarms := FALSE,
                           AdditionalWarnings := FALSE);
   #MachineInterface := "MachineInterface_2_To_1"(MachineInterface_1 := #MachineInterface,
                           MachineInterface_2 := #Orz.MachineInterface,
                           AdditionalAlarms := FALSE,
                           AdditionalWarnings := NOT (NOT #Warning.OP_REST_MissingCnd AND NOT #Warning.OP_WORK_MissingCnd));
END_REGION
END_FUNCTION_BLOCK

FUNCTION "A0302_PareggiatoreCoda_CALL" : Void   // FC138, LAD
// stored: SetENOAutomatically false
BEGIN

REGION Network 1: <<< CIn >>>
END_REGION

REGION Network 2 (SCL): CIn - Trasferimento stati
   REGION TRASFERIMENTO COMANDI CIn MANAGER
       //
       "A0302_PareggiatoreCoda".CIn.Manager := "A0302_Manager".COut.CarroPareggCoda;

   END_REGION
   //
   "A0302_PareggiatoreCoda".CIn.SemiAut_Pb := "A0302_Manager".DataIn.SemiAut_Pb;

   REGION TRASFERIMENTO STATI CIn ALTRE STAZIONI

       // BORDATRICE
       "A0302_PareggiatoreCoda".CIn.Bordatrice.Ax := "A0302_Bordatrice".COut.Ax;

       "A0302_PareggiatoreCoda".CIn.Bordatrice.Sts := "A0302_Bordatrice".COut.Sts;
       "A0302_PareggiatoreCoda".CIn.Bordatrice.RegSpalla.Infeed_ReqON := "A0302_Bordatrice_RegolazioneFormato".Cout.Infeed_ReqON;

       // RULLIERA
       "A0302_PareggiatoreCoda".CIn.Rulliera.Ax_1 := "A0302_Rulliera".COut.Ax_1;
       "A0302_PareggiatoreCoda".CIn.Rulliera.Ax_2 := "A0302_Rulliera".COut.Ax_2;
       "A0302_PareggiatoreCoda".CIn.Rulliera.Centratori := "A0302_Centratori".COut.Centratori;
       "A0302_PareggiatoreCoda".CIn.Rulliera.Coda.Sens.FTC_Rall := "A0302_Rulliera".IEC_FTC_CodaRall.FTC_On;
       "A0302_PareggiatoreCoda".CIn.Rulliera.Coda.Sens.FTC_Prox_Ing := "A0302_Rulliera".IEC_FTC_CodaProxIng.FTC_On;
       "A0302_PareggiatoreCoda".CIn.Rulliera.Centro.Sens.FTC_Centrale := "A0302_Rulliera".IEC_FTC_Centro.FTC_On;

       // CARRO PAREGGIATORE CODA
       "A0302_PareggiatoreCoda".CIn.CarroPareggCoda.Pareggia := "A0302_Manager".Ctrl.TRK.BTrk."Rull-Centratori_TO_Cnd_PareggCoda" OR "A0302_Manager".Ctrl.TRK.BTrk.Cnd_PareggCoda_TO_Pareggiato
       OR "A0302_Manager".Ctrl.CarroPareggCoda.MisuraPzPareggiato;

       // CARRO PAREGGIATORE DI TESTA
       "A0302_PareggiatoreCoda".CIn.CarroPareggTesta.Sens.FTC1_Rall := "A0302_PareggiatoreTesta".IEC_FTC_Rall.FTC_On;
       "A0302_PareggiatoreCoda".CIn.CarroPareggTesta.Sens.FTC2_Prox_Ls := "A0302_PareggiatoreTesta".IEC_FTC_ProxLs.FTC_On;
       "A0302_PareggiatoreCoda".CIn.CarroPareggTesta.Sens.PresenzaMat := "A0302_PareggiatoreTesta".IEC_FTC_PresentMat.FTC_On;

       // STATI DELLA STAZIONE 
       "A0302_PareggiatoreCoda".CIn.CarriPareggiatori.ZoneA0302Entry_Empty := "A0302_Manager".Sts.BTrk.ZoneA0302Entry_Empty;
       "A0302_PareggiatoreCoda".CIn.CarriPareggiatori.ZoneA0302Exit_Empty := "A0302_Manager".Sts.BTrk.ZoneA0302Exit_Empty;
       "A0302_PareggiatoreCoda".CIn.CarriPareggiatori.RequestNewPosition := "A0302_Manager".Sts.Attrezzamento.RequestNewPosition;

       // SPALLE
       "A0302_PareggiatoreCoda".CIn.Spalle.Coda.ActualPos := "Areas_ITF".A04.A0303_SpallaCoda_Cout_Ax.ActualPosition;
       "A0302_PareggiatoreCoda".CIn.Spalle.Testa.ActualPos := "Areas_ITF".A04.A0303_SpallaTesta_Cout_Ax.ActualPosition;

       // MANIPOLATORE
       "A0302_PareggiatoreCoda".CIn.Manipolatore.Sollevatore := "A0302_Manipolatore".COut.Coda.Sollevatore;

       // CENTRATORE
       "A0302_PareggiatoreCoda".CIn.Centratori.Sollevamento := "A0302_Centratori".COut.Sollevamento;

   END_REGION ;
END_REGION

REGION Network 3: CIn Oil In Pressure
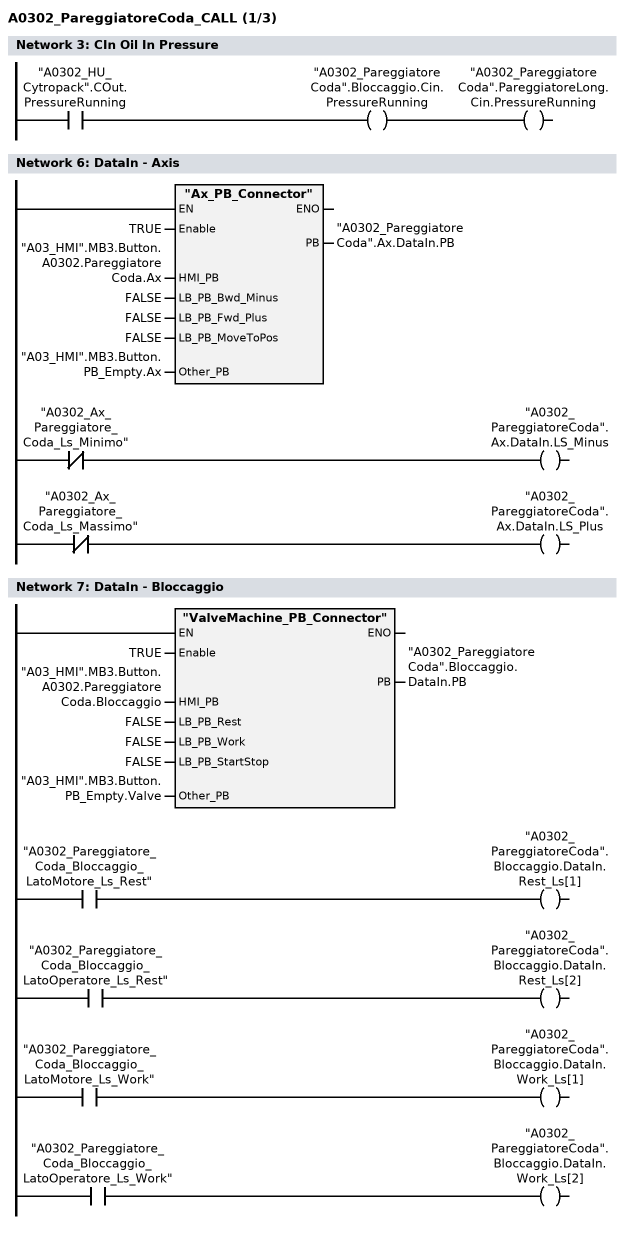
   RUNG wire#powerrail
      Contact( "A0302_HU_Cytropack".COut.PressureRunning )
      Coil( "A0302_PareggiatoreCoda".Bloccaggio.Cin.PressureRunning )
      Coil( "A0302_PareggiatoreCoda".PareggiatoreLong.Cin.PressureRunning )
   END_RUNG
   // the same network as SCL:
   "A0302_PareggiatoreCoda".Bloccaggio.Cin.PressureRunning := "A0302_HU_Cytropack".COut.PressureRunning;
   "A0302_PareggiatoreCoda".PareggiatoreLong.Cin.PressureRunning := "A0302_HU_Cytropack".COut.PressureRunning;
END_REGION

REGION Network 4: <<< DATA IN >>>
END_REGION

REGION Network 5 (SCL): DataIn - OP e sensori

   REGION TRASFERIMENTO DATA In
       // Pulsanti OP lavoro
       "A0302_PareggiatoreCoda".DataIn.BattutaVrt.OP.Rest := "A03_HMI".MB3.Button.A0302.PareggiatoreCoda.OP_BattutaVrt.Rest;
       "A0302_PareggiatoreCoda".DataIn.BattutaVrt.OP.Work := "A03_HMI".MB3.Button.A0302.PareggiatoreCoda.OP_BattutaVrt.Work;
       "A0302_PareggiatoreCoda".DataIn.PareggLong.OP.Rest := "A03_HMI".MB3.Button.A0302.PareggiatoreCoda.OP_PareggLong.Rest;
       "A0302_PareggiatoreCoda".DataIn.PareggLong.OP.Work := "A03_HMI".MB3.Button.A0302.PareggiatoreCoda.OP_PareggLong.Work;
       "A0302_PareggiatoreCoda".DataIn.OP_MoveToPos := "A0302_PareggiatoreCoda".Ax.DataIn.PB.MoveToPos;

       // Ingressi Sensori
       "A0302_PareggiatoreCoda".DataIn.PareggLong.AnalSens := "A0302_AI_Pareggiatore_Coda_Longitudinale_Posizionamento"; 

       // FTC pezzo in arrivo
       "A0302_PareggiatoreCoda".DataIn.Sens.FTC_Ingombro_In := "A0302_Rulliera_Lato_2_Coda_Phc_PezzoInArrivo";
       // FTC pezzo dopo battuta coda
       "A0302_PareggiatoreCoda".DataIn.Sens.FTC_Ingombro_Out := "A0302_Rulliera_Lato_2_Coda_Phc_PezzoDopoBattuta";
       // FTC presenza materiale su manipolatori
       "A0302_PareggiatoreCoda".DataIn.Sens.PresenzaMat := "A0302_Manipolatore_Coda_Magnete_Ls_Work";


       // Extracorsa Pareggiatore testa
       "A0302_PareggiatoreCoda".DataIn.Sens.FC_Aticoll_Spalla := NOT "A0302_Ax_Pareggiatore_Coda_AntiCollisione";

   END_REGION ;
END_REGION

REGION Network 6: DataIn - Axis
   RUNG wire#powerrail
      "Ax_PB_Connector"(Enable := TRUE, HMI_PB := "A03_HMI".MB3.Button.A0302.PareggiatoreCoda.Ax, LB_PB_Bwd_Minus := FALSE, LB_PB_Fwd_Plus := FALSE, LB_PB_MoveToPos := FALSE, Other_PB := "A03_HMI".MB3.Button.PB_Empty.Ax, PB => "A0302_PareggiatoreCoda".Ax.DataIn.PB)
   END_RUNG
   RUNG wire#powerrail
      I_Contact( "A0302_Ax_Pareggiatore_Coda_Ls_Minimo" )
      Coil( "A0302_PareggiatoreCoda".Ax.DataIn.LS_Minus )
   END_RUNG
   RUNG wire#powerrail
      I_Contact( "A0302_Ax_Pareggiatore_Coda_Ls_Massimo" )
      Coil( "A0302_PareggiatoreCoda".Ax.DataIn.LS_Plus )
   END_RUNG
   // the same network as SCL:
   "Ax_PB_Connector"(Enable := TRUE,
                     HMI_PB := "A03_HMI".MB3.Button.A0302.PareggiatoreCoda.Ax,
                     LB_PB_Bwd_Minus := FALSE,
                     LB_PB_Fwd_Plus := FALSE,
                     LB_PB_MoveToPos := FALSE,
                     Other_PB := "A03_HMI".MB3.Button.PB_Empty.Ax,
                     PB => "A0302_PareggiatoreCoda".Ax.DataIn.PB);
   "A0302_PareggiatoreCoda".Ax.DataIn.LS_Minus := NOT "A0302_Ax_Pareggiatore_Coda_Ls_Minimo";
   "A0302_PareggiatoreCoda".Ax.DataIn.LS_Plus := NOT "A0302_Ax_Pareggiatore_Coda_Ls_Massimo";
END_REGION

REGION Network 7: DataIn - Bloccaggio
   RUNG wire#powerrail
      "ValveMachine_PB_Connector"(Enable := TRUE, HMI_PB := "A03_HMI".MB3.Button.A0302.PareggiatoreCoda.Bloccaggio, LB_PB_Rest := FALSE, LB_PB_Work := FALSE, LB_PB_StartStop := FALSE, Other_PB := "A03_HMI".MB3.Button.PB_Empty.Valve, PB => "A0302_PareggiatoreCoda".Bloccaggio.DataIn.PB)
   END_RUNG
   RUNG wire#powerrail
      Contact( "A0302_Pareggiatore_Coda_Bloccaggio_LatoMotore_Ls_Rest" )
      Coil( "A0302_PareggiatoreCoda".Bloccaggio.DataIn.Rest_Ls[1] )
   END_RUNG
   RUNG wire#powerrail
      Contact( "A0302_Pareggiatore_Coda_Bloccaggio_LatoOperatore_Ls_Rest" )
      Coil( "A0302_PareggiatoreCoda".Bloccaggio.DataIn.Rest_Ls[2] )
   END_RUNG
   RUNG wire#powerrail
      Contact( "A0302_Pareggiatore_Coda_Bloccaggio_LatoMotore_Ls_Work" )
      Coil( "A0302_PareggiatoreCoda".Bloccaggio.DataIn.Work_Ls[1] )
   END_RUNG
   RUNG wire#powerrail
      Contact( "A0302_Pareggiatore_Coda_Bloccaggio_LatoOperatore_Ls_Work" )
      Coil( "A0302_PareggiatoreCoda".Bloccaggio.DataIn.Work_Ls[2] )
   END_RUNG
   // the same network as SCL:
   "ValveMachine_PB_Connector"(Enable := TRUE,
                           HMI_PB := "A03_HMI".MB3.Button.A0302.PareggiatoreCoda.Bloccaggio,
                           LB_PB_Rest := FALSE,
                           LB_PB_Work := FALSE,
                           LB_PB_StartStop := FALSE,
                           Other_PB := "A03_HMI".MB3.Button.PB_Empty.Valve,
                           PB => "A0302_PareggiatoreCoda".Bloccaggio.DataIn.PB);
   "A0302_PareggiatoreCoda".Bloccaggio.DataIn.Rest_Ls[1] := "A0302_Pareggiatore_Coda_Bloccaggio_LatoMotore_Ls_Rest";
   "A0302_PareggiatoreCoda".Bloccaggio.DataIn.Rest_Ls[2] := "A0302_Pareggiatore_Coda_Bloccaggio_LatoOperatore_Ls_Rest";
   "A0302_PareggiatoreCoda".Bloccaggio.DataIn.Work_Ls[1] := "A0302_Pareggiatore_Coda_Bloccaggio_LatoMotore_Ls_Work";
   "A0302_PareggiatoreCoda".Bloccaggio.DataIn.Work_Ls[2] := "A0302_Pareggiatore_Coda_Bloccaggio_LatoOperatore_Ls_Work";
END_REGION

REGION Network 8: DataIn - Battuta Verticale
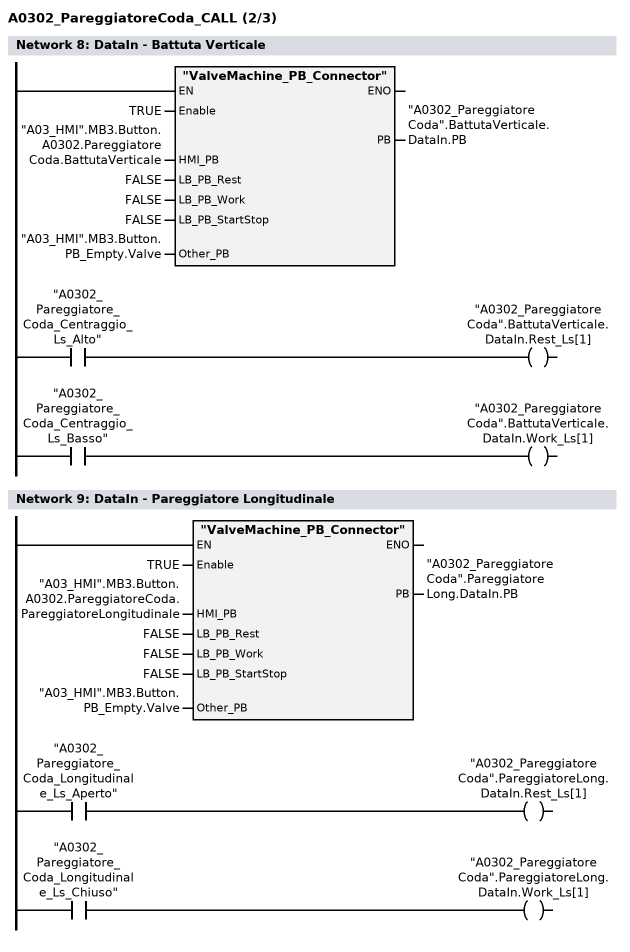
   RUNG wire#powerrail
      "ValveMachine_PB_Connector"(Enable := TRUE, HMI_PB := "A03_HMI".MB3.Button.A0302.PareggiatoreCoda.BattutaVerticale, LB_PB_Rest := FALSE, LB_PB_Work := FALSE, LB_PB_StartStop := FALSE, Other_PB := "A03_HMI".MB3.Button.PB_Empty.Valve, PB => "A0302_PareggiatoreCoda".BattutaVerticale.DataIn.PB)
   END_RUNG
   RUNG wire#powerrail
      Contact( "A0302_Pareggiatore_Coda_Centraggio_Ls_Alto" )
      Coil( "A0302_PareggiatoreCoda".BattutaVerticale.DataIn.Rest_Ls[1] )
   END_RUNG
   RUNG wire#powerrail
      Contact( "A0302_Pareggiatore_Coda_Centraggio_Ls_Basso" )
      Coil( "A0302_PareggiatoreCoda".BattutaVerticale.DataIn.Work_Ls[1] )
   END_RUNG
   // the same network as SCL:
   "ValveMachine_PB_Connector"(Enable := TRUE,
                           HMI_PB := "A03_HMI".MB3.Button.A0302.PareggiatoreCoda.BattutaVerticale,
                           LB_PB_Rest := FALSE,
                           LB_PB_Work := FALSE,
                           LB_PB_StartStop := FALSE,
                           Other_PB := "A03_HMI".MB3.Button.PB_Empty.Valve,
                           PB => "A0302_PareggiatoreCoda".BattutaVerticale.DataIn.PB);
   "A0302_PareggiatoreCoda".BattutaVerticale.DataIn.Rest_Ls[1] := "A0302_Pareggiatore_Coda_Centraggio_Ls_Alto";
   "A0302_PareggiatoreCoda".BattutaVerticale.DataIn.Work_Ls[1] := "A0302_Pareggiatore_Coda_Centraggio_Ls_Basso";
END_REGION

REGION Network 9: DataIn - Pareggiatore Longitudinale
   RUNG wire#powerrail
      "ValveMachine_PB_Connector"(Enable := TRUE, HMI_PB := "A03_HMI".MB3.Button.A0302.PareggiatoreCoda.PareggiatoreLongitudinale, LB_PB_Rest := FALSE, LB_PB_Work := FALSE, LB_PB_StartStop := FALSE, Other_PB := "A03_HMI".MB3.Button.PB_Empty.Valve, PB => "A0302_PareggiatoreCoda".PareggiatoreLong.DataIn.PB)
   END_RUNG
   RUNG wire#powerrail
      Contact( "A0302_Pareggiatore_Coda_Longitudinale_Ls_Aperto" )
      Coil( "A0302_PareggiatoreCoda".PareggiatoreLong.DataIn.Rest_Ls[1] )
   END_RUNG
   RUNG wire#powerrail
      Contact( "A0302_Pareggiatore_Coda_Longitudinale_Ls_Chiuso" )
      Coil( "A0302_PareggiatoreCoda".PareggiatoreLong.DataIn.Work_Ls[1] )
   END_RUNG
   // the same network as SCL:
   "ValveMachine_PB_Connector"(Enable := TRUE,
                           HMI_PB := "A03_HMI".MB3.Button.A0302.PareggiatoreCoda.PareggiatoreLongitudinale,
                           LB_PB_Rest := FALSE,
                           LB_PB_Work := FALSE,
                           LB_PB_StartStop := FALSE,
                           Other_PB := "A03_HMI".MB3.Button.PB_Empty.Valve,
                           PB => "A0302_PareggiatoreCoda".PareggiatoreLong.DataIn.PB);
   "A0302_PareggiatoreCoda".PareggiatoreLong.DataIn.Rest_Ls[1] := "A0302_Pareggiatore_Coda_Longitudinale_Ls_Aperto";
   "A0302_PareggiatoreCoda".PareggiatoreLong.DataIn.Work_Ls[1] := "A0302_Pareggiatore_Coda_Longitudinale_Ls_Chiuso";
END_REGION

REGION Network 10: <+>
END_REGION

REGION Network 11 (SCL): Drive
   "A0302_PareggiatoreCoda".Drive.Infeed_ON := "Areas_ITF".AG.Infeed_Running;;
   "A0302_PareggiatoreCoda".Drive.AccessPoint := "HW_Const_Values".CU6_PN_605A1_ModuleAccessPoint;
   "A0302_PareggiatoreCoda".Drive.AxisID := "CU6_ID_5_2100A1_2_2180M1";
   "A0302_PareggiatoreCoda".Drive.TokenChain := "TOKENCHAIN_CU6";
END_REGION

REGION Network 12 (SCL): HW
   "A0302_PareggiatoreCoda".HWID.Ax_TEL1 :="HW_Const_Values".CU6_PN_2100A1_2_Standard_telegram_1 ;
   "A0302_PareggiatoreCoda".HWID.Enc_IO := "HW_Const_Values".HW_2184P1_Telegram_81_DI_DO;
END_REGION

REGION Network 13: [Pareggiatore Coda FB] - Machine Call
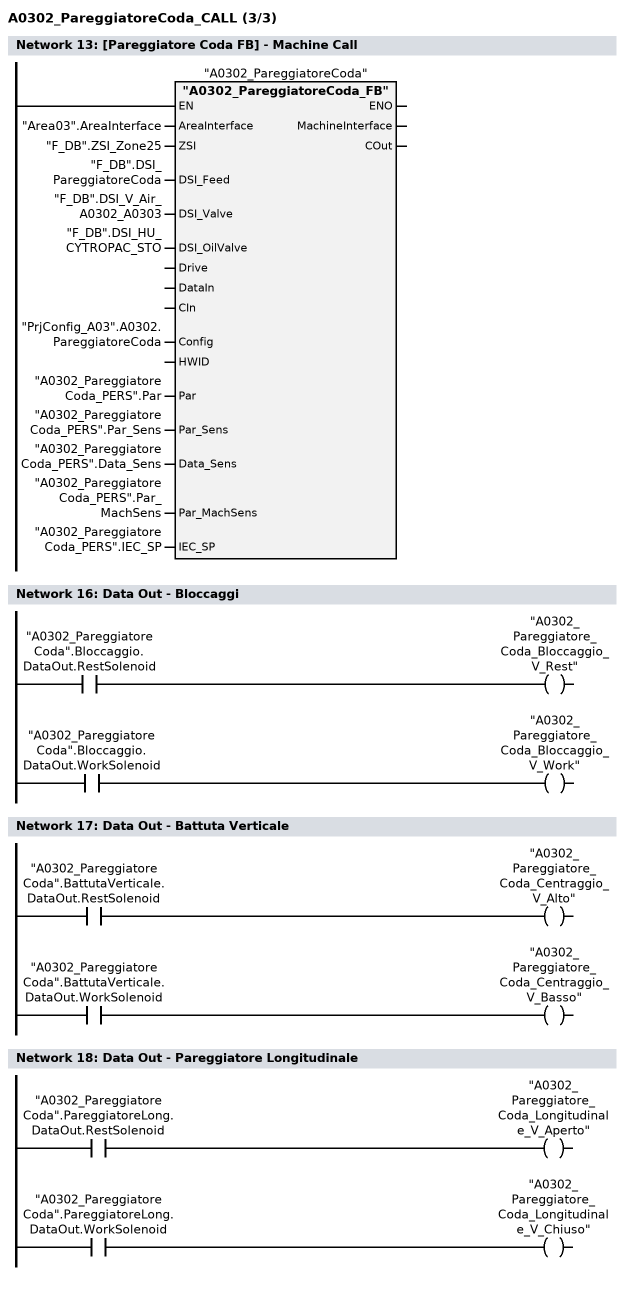
   RUNG wire#powerrail
      "A0302_PareggiatoreCoda"(AreaInterface := "Area03".AreaInterface, ZSI := "F_DB".ZSI_Zone25, DSI_Feed := "F_DB".DSI_PareggiatoreCoda, DSI_Valve := "F_DB".DSI_V_Air_A0302_A0303, DSI_OilValve := "F_DB".DSI_HU_CYTROPAC_STO, Drive :=, DataIn :=, CIn :=, Config := "PrjConfig_A03".A0302.PareggiatoreCoda, HWID :=, Par := "A0302_PareggiatoreCoda_PERS".Par, Par_Sens := "A0302_PareggiatoreCoda_PERS".Par_Sens, Data_Sens := "A0302_PareggiatoreCoda_PERS".Data_Sens, Par_MachSens := "A0302_PareggiatoreCoda_PERS".Par_MachSens, IEC_SP := "A0302_PareggiatoreCoda_PERS".IEC_SP, MachineInterface =>, COut =>)
   END_RUNG
   // the same network as SCL:
   "A0302_PareggiatoreCoda"(AreaInterface := "Area03".AreaInterface,   // "A0302_PareggiatoreCoda_FB"
                           ZSI := "F_DB".ZSI_Zone25,
                           DSI_Feed := "F_DB".DSI_PareggiatoreCoda,
                           DSI_Valve := "F_DB".DSI_V_Air_A0302_A0303,
                           DSI_OilValve := "F_DB".DSI_HU_CYTROPAC_STO,
                           Config := "PrjConfig_A03".A0302.PareggiatoreCoda,
                           Par := "A0302_PareggiatoreCoda_PERS".Par,
                           Par_Sens := "A0302_PareggiatoreCoda_PERS".Par_Sens,
                           Data_Sens := "A0302_PareggiatoreCoda_PERS".Data_Sens,
                           Par_MachSens := "A0302_PareggiatoreCoda_PERS".Par_MachSens,
                           IEC_SP := "A0302_PareggiatoreCoda_PERS".IEC_SP);
END_REGION

REGION Network 15: <<< DATA OUT >>>
END_REGION

REGION Network 16: Data Out - Bloccaggi
   RUNG wire#powerrail
      Contact( "A0302_PareggiatoreCoda".Bloccaggio.DataOut.RestSolenoid )
      Coil( "A0302_Pareggiatore_Coda_Bloccaggio_V_Rest" )
   END_RUNG
   RUNG wire#powerrail
      Contact( "A0302_PareggiatoreCoda".Bloccaggio.DataOut.WorkSolenoid )
      Coil( "A0302_Pareggiatore_Coda_Bloccaggio_V_Work" )
   END_RUNG
   // the same network as SCL:
   "A0302_Pareggiatore_Coda_Bloccaggio_V_Rest" := "A0302_PareggiatoreCoda".Bloccaggio.DataOut.RestSolenoid;
   "A0302_Pareggiatore_Coda_Bloccaggio_V_Work" := "A0302_PareggiatoreCoda".Bloccaggio.DataOut.WorkSolenoid;
END_REGION

REGION Network 17: Data Out - Battuta Verticale
   RUNG wire#powerrail
      Contact( "A0302_PareggiatoreCoda".BattutaVerticale.DataOut.RestSolenoid )
      Coil( "A0302_Pareggiatore_Coda_Centraggio_V_Alto" )
   END_RUNG
   RUNG wire#powerrail
      Contact( "A0302_PareggiatoreCoda".BattutaVerticale.DataOut.WorkSolenoid )
      Coil( "A0302_Pareggiatore_Coda_Centraggio_V_Basso" )
   END_RUNG
   // the same network as SCL:
   "A0302_Pareggiatore_Coda_Centraggio_V_Alto" := "A0302_PareggiatoreCoda".BattutaVerticale.DataOut.RestSolenoid;
   "A0302_Pareggiatore_Coda_Centraggio_V_Basso" := "A0302_PareggiatoreCoda".BattutaVerticale.DataOut.WorkSolenoid;
END_REGION

REGION Network 18: Data Out - Pareggiatore Longitudinale
   RUNG wire#powerrail
      Contact( "A0302_PareggiatoreCoda".PareggiatoreLong.DataOut.RestSolenoid )
      Coil( "A0302_Pareggiatore_Coda_Longitudinale_V_Aperto" )
   END_RUNG
   RUNG wire#powerrail
      Contact( "A0302_PareggiatoreCoda".PareggiatoreLong.DataOut.WorkSolenoid )
      Coil( "A0302_Pareggiatore_Coda_Longitudinale_V_Chiuso" )
   END_RUNG
   // the same network as SCL:
   "A0302_Pareggiatore_Coda_Longitudinale_V_Aperto" := "A0302_PareggiatoreCoda".PareggiatoreLong.DataOut.RestSolenoid;
   "A0302_Pareggiatore_Coda_Longitudinale_V_Chiuso" := "A0302_PareggiatoreCoda".PareggiatoreLong.DataOut.WorkSolenoid;
END_REGION
END_FUNCTION

FUNCTION_BLOCK "A0302_PareggiatoreCoda_FB"   // FB118, LAD
// stored: MemoryReserve 100, SetENOAutomatically false
   VAR_INPUT
      AreaInterface : "AreaInterface";
      ZSI : "udt_ZoneSafetyInterface";
      DSI_Feed : "udt_DeviceSafetyInterface";
      DSI_Valve : "udt_DeviceSafetyInterface";
      DSI_OilValve : "udt_DeviceSafetyInterface";
      Drive : "TAx_DriveInterface";
      DataIn : Struct
         OP_MoveToPos : Bool;
         BattutaVrt : Struct
            OP : "OP_PB";
         END_STRUCT;
         PareggLong : Struct
            OP : "OP_PB";
            AnalSens : Int;
         END_STRUCT;
         Sens { ExternalWritable := 'False'} : Struct
            FTC_Ingombro_In : Bool;   // 2012BF1 - I50.0
            FTC_Ingombro_Out : Bool;   // 2012BF2 - I50.1
            PresenzaMat : Bool;   // FC presenza materiale agganciato lato paregg coda
            FC_Aticoll_Spalla : Bool;
         END_STRUCT;
      END_STRUCT;
      CIn : Struct
         Manager : Struct
            EnableStopDoorOpeningReq { ExternalAccessible := 'False'; ExternalVisible := 'False'; ExternalWritable := 'False'} : Bool;
            EnableStopInPhase { ExternalAccessible := 'False'; ExternalVisible := 'False'; ExternalWritable := 'False'} : Bool;
            EnableStopProgrammed { ExternalAccessible := 'False'; ExternalVisible := 'False'; ExternalWritable := 'False'} : Bool;
            Control_ON { ExternalAccessible := 'False'; ExternalVisible := 'False'; ExternalWritable := 'False'} : Bool;
            MoveToPos { ExternalAccessible := 'False'; ExternalVisible := 'False'; ExternalWritable := 'False'} : Bool;
            Pos { ExternalAccessible := 'False'; ExternalVisible := 'False'; ExternalWritable := 'False'} : LReal;
            Speed : LReal;
            Bloccaggio { ExternalAccessible := 'False'; ExternalVisible := 'False'; ExternalWritable := 'False'} : Struct
               Rest : Bool;
               Work : Bool;
            END_STRUCT;
            BattutaVrt { ExternalAccessible := 'False'; ExternalVisible := 'False'; ExternalWritable := 'False'} : Struct
               Rest : Bool;
               Work : Bool;
            END_STRUCT;
            PareggLong { ExternalAccessible := 'False'; ExternalVisible := 'False'; ExternalWritable := 'False'} : Struct
               Rest : Bool;
               Work : Bool;
            END_STRUCT;
         END_STRUCT;
         SemiAut_Pb { ExternalWritable := 'False'} : Bool;
         Bordatrice : Struct
            Ax : "Positioning_EPOS_Machine_COut";
            Sts : Struct
               PosTargetEnable : Bool;
               PosTarget_Reached : Bool;
               In_W_Pos : Bool;
               AtRest : Bool;
            END_STRUCT;
            RegSpalla : Struct
               Infeed_ReqON : Bool;
            END_STRUCT;
         END_STRUCT;
         Rulliera { ExternalWritable := 'False'} : Struct
            Ax_1 : "SpeedMachine_COut";
            Ax_2 : "SpeedMachine_COut";
            Centratori : "ValveMachine_COut";
            Coda : Struct
               Sens : Struct
                  FTC_Rall : Bool;   // Sensori presenza materiale banco rallentamento ingresso
                  FTC_Prox_Ing : Bool;   // Sensori presenza materiale banco limite ingresso
               END_STRUCT;
            END_STRUCT;
            Centro : Struct
               Sens : Struct
                  FTC_Centrale : Bool;   // 2010BF1 - I50.2
               END_STRUCT;
            END_STRUCT;
         END_STRUCT;
         CarroPareggCoda : Struct
            Pareggia : Bool;   // Bit di abilitazione pareggiamento - prende la misura del beam e controlla la tolleranza
            OilInTargetPressure { ExternalWritable := 'False'} : Bool;
         END_STRUCT;
         CarroPareggTesta { ExternalWritable := 'False'} : Struct
            Sens : Struct
               FTC1_Rall : Bool;   // 2010BF2 - I50.3
               FTC2_Prox_Ls : Bool;   // 2010BF3 - I50.4
               PresenzaMat : Bool;   // FC presenza materiale agganciato lato paregg testa
            END_STRUCT;
         END_STRUCT;
         CarriPareggiatori : Struct
            ZoneA0302Entry_Empty { ExternalWritable := 'False'} : Bool;
            ZoneA0302Exit_Empty { ExternalWritable := 'False'} : Bool;
            RequestNewPosition : Bool;
         END_STRUCT;
         Spalle : Struct
            Coda : Struct
               ActualPos : LReal;
            END_STRUCT;
            Testa : Struct
               ActualPos : LReal;
            END_STRUCT;
         END_STRUCT;
         Manipolatore : Struct
            Sollevatore : "ValveMachine_COut";
         END_STRUCT;
         Centratori : Struct
            Sollevamento : "ValveMachine_COut";
         END_STRUCT;
      END_STRUCT;
      Config : Struct
         Ax : "Positioning_DOL_Machine_Config";
         Bloccaggio : "ValveMachine_Config";
         BattutaVerticale : "ValveMachine_Config";
         PareggiatoreLong : "ValveMachine_Config";
         PosPareggiatore : Struct
            QuotaMin_Work : LReal;
            QuotaMax_Work : LReal;
         END_STRUCT;
         MinDistanzaConSpalla : LReal;
         DelayMissingCondition : Time;
      END_STRUCT;
      HWID : Struct
         Ax_TEL1 : HW_SUBMODULE;
         Enc_IO : HW_SUBMODULE;
      END_STRUCT;
   END_VAR
   VAR_OUTPUT
      MachineInterface : "MachineInterface";
      COut : Struct
         Ax : "Positioning_DOL_Machine_COut";
         Bloccaggio : "ValveMachine_COut";
         BattutaVerticale : "ValveMachine_COut";
         PareggiatoreLong : "ValveMachine_COut";
         Ax_InWPos : Bool;
         Anticipi : Struct
            Work : Struct
               BattutaVrt : Bool;
               PareggLong : Bool;
            END_STRUCT;
            Rest : Struct
               BattutaVrt : Bool;
               PareggLong : Bool;
            END_STRUCT;
         END_STRUCT;
      END_STRUCT;
   END_VAR
   VAR_IN_OUT
      Par : Struct
         Ax : "Positioning_DOL_Machine_Par";
         Ax_Pers : "Positioning_DOL_Machine_Pers_Data";
         Enc : "PosFbk_RTN";
         Ax_Aut : "A0301_Mach_Speed_Par";
         Bloccaggio_Sens : Struct
            "2191B1" : "Analogic_SensorManagement_Par";
            SogliaWork : Real;
         END_STRUCT;
         CarroPareggCoda : Struct
            Delay_StartMove : Time;
            Preset : LReal;
         END_STRUCT;
         Cremaliera : Struct
            Modulo : LReal;
            Passo : LReal;
         END_STRUCT;
      END_STRUCT;
      Par_Sens : Struct
         AI : "Analogic_SensorManagement_Par";
      END_STRUCT;
      Data_Sens : "Analogic_SensorManagement_Data";
      Par_MachSens : "A0301_Mach_Sens_Par";
      IEC_SP : Struct
         FTC_Input : Struct
            TON_PT : Time;
            TOF_PT : Time;
         END_STRUCT;
         FTC_Output : Struct
            TON_PT : Time;
            TOF_PT : Time;
         END_STRUCT;
         FTC_PresentMat : Struct
            TON_PT : Time;
            TOF_PT : Time;
         END_STRUCT;
         Check_2119B1 : Struct
            TON_PT : Time;
         END_STRUCT;
      END_STRUCT;
   END_VAR
   VAR
      Alarm : Struct
         Ax : "Positioning_DOL_Machine_Alr";
         Enc : "PosFbk_Encoder_Alr";
         Bloccaggio : "ValveAlr";
         BattutaVerticale : "ValveAlr";
         PareggiatoreLong : "ValveAlr";
         PareggLong_AnalSens_Issue : Bool;
         SensFC_Aticoll_Spalla : Bool;
         Bloccaggio_AnalSens_Issue : Bool;   // Errore soglia lettura pressione su bloccaggio cremaliera
      END_STRUCT;
      Warning : Struct
         Ax : "Positioning_DOL_Machine_Wng";
         Bloccaggio : "ValveMachine_Wng";
         BattutaVerticale : "ValveMachine_Wng";
         PareggiatoreLongitudinale : "ValveMachine_Wng";
         PosPareggiatoreLong : "Analogic_SensorManagement_Warning";
         MissingCnd : Struct
            OP_REST_BattutaVrt : Bool;   // Mancanza comando arresto
            OP_WORK_BattutaVrt : Bool;   // Mancanza consenso lavoro
            OP_REST_PareggLong : Bool;   // Mancanza comando arresto
            OP_WORK_PareggLong : Bool;   // Mancanza consenso lavoro
            OP_REST_Bloccaggio : Bool;   // Mancanza comando arresto
            OP_WORK_Bloccaggio : Bool;   // Mancanza consenso lavoro
         END_STRUCT;
         SW_Limit_AntiCollision : Bool;
      END_STRUCT;
      HMI : Struct
         AnalogSensor : "AnalogSens_HmiData";
         Ax : Struct
            PbPreset : Bool;
            B_Preset_UM2 : Bool;
            PresetValue : LReal;
         END_STRUCT;
      END_STRUCT;
      Sts : Struct
         ReadyForMove : Bool;   // Pronto al movimento
         OP_PCoda_CanMoveFreely : Bool;
         OP_Ax_CanMoveFreely : Bool;
         Op_MoveToPos_Cnd : Bool;
         BattutaVrt : Struct
            OP_Rest_Cnd : Bool;
            Op_Work_Cnd : Bool;
         END_STRUCT;
         PareggLong : Struct
            OP_Rest_Cnd : Bool;
            Op_Work_Cnd : Bool;
         END_STRUCT;
      END_STRUCT;
      Ctrl : Struct
         BattutaVrt : Struct
            OP_Rest_Man : Bool;
            OP_Work_Man : Bool;
            OP_Rest_Aut : Bool;
            OP_Work_Aut : Bool;
            OP_Rest : Bool;
            OP_Work : Bool;
         END_STRUCT;
         PareggLong : Struct
            CheckMesure : Bool;   // Bit che determina l'uscita del pareggiatore e Controlla misura Blea nel manager
            OP_Rest_Aut : Bool;
            OP_Work_Aut : Bool;
            OP_Rest_Man : Bool;
            OP_Work_Man : Bool;
            OP_Rest : Bool;
            OP_Work : Bool;
         END_STRUCT;
         Ax : Struct
            OP_MoveToPos_Man : Bool;
            OP_MoveToPos_Aut : Bool;
            OP_MoveToPos : Bool;
         END_STRUCT;
      END_STRUCT;
      AUX : Struct
         OP_MoveToPos : Bool;
         BattutaVrt : Struct
            OP_Rest : Bool;
            OP_Work : Bool;
         END_STRUCT;
         PareggLong : Struct
            OP_Rest : Bool;
            OP_Work : Bool;
         END_STRUCT;
      END_STRUCT;
      Ax { S7_SetPoint := 'True'} : "Positioning_DOL_Machine_FB";   // Asse di movimento carro pareggiatore su cremaliera
      Enc : "PosFbk_SickAFM60";
      Enc_ITF : "PosFbk_ITF";
      Bloccaggio { S7_SetPoint := 'True'} : "ValveMachine_FB";   // Bloccaggio cremaliera
      BattutaVerticale { S7_SetPoint := 'True'} : "ValveMachine_FB";   // Battuta verticale
      PareggiatoreLong { S7_SetPoint := 'True'} : "ValveMachine_FB";   // Pareggiatore longitudinale
      PosPareggLong { S7_SetPoint := 'True'} : "Analogic_SensorManagement";   // Sensore di posizione pareggiatore
      TON_PareggLong : Struct
         OP_REST_MissingCnd { S7_SetPoint := 'True'} : TON_TIME;
         OP_WORK_MissingCnd { S7_SetPoint := 'True'} : TON_TIME;
      END_STRUCT;
      TON_BattutaVrt : Struct
         OP_REST_MissingCnd { S7_SetPoint := 'True'} : TON_TIME;
         OP_WORK_MissingCnd { S7_SetPoint := 'True'} : TON_TIME;
      END_STRUCT;
      TON_Bloccaggio : Struct
         OP_REST_MissingCnd { S7_SetPoint := 'True'} : TON_TIME;
         OP_WORK_MissingCnd { S7_SetPoint := 'True'} : TON_TIME;
      END_STRUCT;
      IEC_FTC_Input : Struct
         TON_Delay : IEC_TIMER;
         TOF_Delay { S7_SetPoint := 'True'} : IEC_TIMER;
         FTC_On { S7_SetPoint := 'True'} : Bool;
      END_STRUCT;
      IEC_FTC_Output : Struct
         TON_Delay : IEC_TIMER;
         TOF_Delay { S7_SetPoint := 'True'} : IEC_TIMER;
         FTC_On { S7_SetPoint := 'True'} : Bool;
      END_STRUCT;
      IEC_FTC_PresentMat : Struct
         TON_Delay : IEC_TIMER;
         TOF_Delay { S7_SetPoint := 'True'} : IEC_TIMER;
         FTC_On { S7_SetPoint := 'True'} : Bool;
      END_STRUCT;
      IEC_DelayCheck_2119B1 : IEC_TIMER;
      Bloccaggio_AnalSens { S7_SetPoint := 'True'} : "AnalogThreshold";
      CarroCoda { ExternalAccessible := 'False'; ExternalVisible := 'False'; ExternalWritable := 'False'} : Struct
         RimanenzaPos : LReal;
         PassoReq : LReal;
         PosBattutePz : LReal;
         SemiBeamLen : LReal;
         NrPassiReq : LReal;
         Pos : LReal;   // Posizione calcolata in funzione della cremaliera
      END_STRUCT;
      TON_DistanzaOK : IEC_TIMER;
      TON_Anticipi : Struct
         Rest : Struct
            BattutaVrt { S7_SetPoint := 'True'} : IEC_TIMER;
            PareggLong : IEC_TIMER;
         END_STRUCT;
         Work : Struct
            PareggLong : IEC_TIMER;
            BattutaVrt { S7_SetPoint := 'True'} : IEC_TIMER;
         END_STRUCT;
      END_STRUCT;
   END_VAR
   VAR_TEMP
      PE : Struct
         OP_MoveToPos : Bool;
         BattutaVrt : Struct
            OP_Rest : Bool;
            OP_Work : Bool;
         END_STRUCT;
         PareggLong : Struct
            OP_Rest : Bool;
            OP_Work : Bool;
         END_STRUCT;
      END_STRUCT;
      ActualDifference : LReal;
   END_VAR
   VAR CONSTANT
      RACK_STEP : LReal;   // Passo Cremagliera mm
   END_VAR
   VAR_TEMP   // added for the SCL form of the ladder/FBD networks
      _w1 : Bool;
      _w2 : Bool;
      _w3 : Bool;
      _w4 : Bool;
      _w5 : Bool;
      _w6 : Bool;
      _w7 : Bool;
      _w8 : Bool;
      _w9 : Bool;
      _w10 : Bool;
      _w11 : Bool;
      _w12 : Bool;
   END_VAR
BEGIN

REGION Network 1 (SCL): Reset allarmi
   IF #AreaInterface.RstAlarms THEN
       #Alarm.PareggLong_AnalSens_Issue := FALSE;
       #Alarm.SensFC_Aticoll_Spalla := FALSE;
       #Alarm.Bloccaggio_AnalSens_Issue := FALSE;
   END_IF;
END_REGION

REGION Network 2: <+>
END_REGION

REGION Network 3: Anticipi Movimento LAVORO
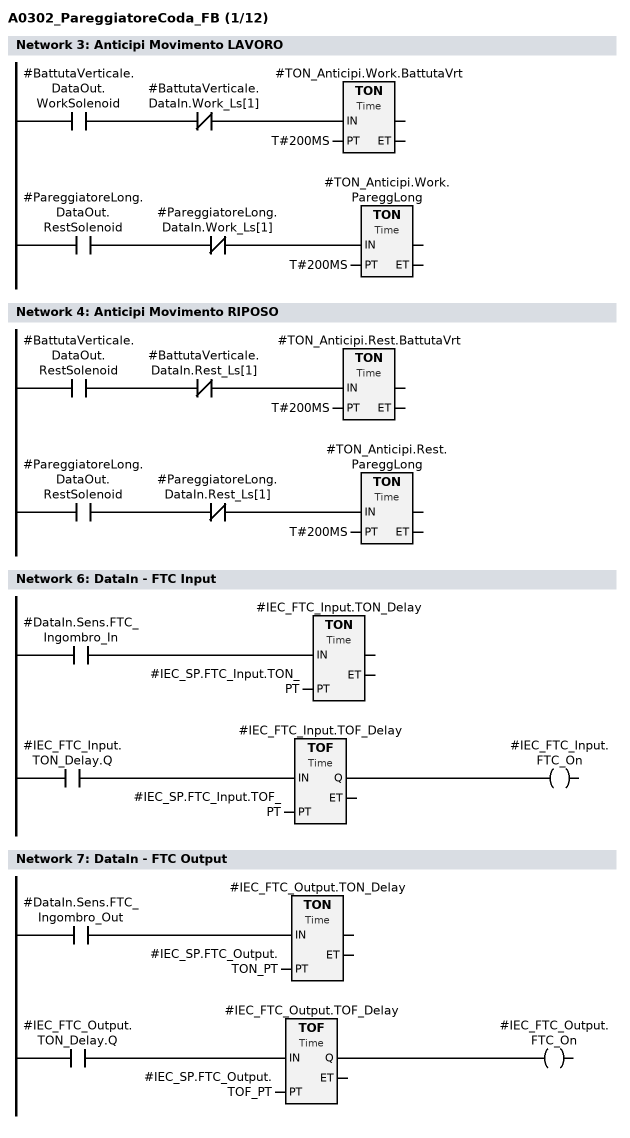
   RUNG wire#powerrail
      Contact( #BattutaVerticale.DataOut.WorkSolenoid )
      I_Contact( #BattutaVerticale.DataIn.Work_Ls[1] )
      { S7_Templates := "time_type := Time" } #TON_Anticipi.Work.BattutaVrt.TON(pt := T#200MS, et =>)
   END_RUNG
   RUNG wire#powerrail
      Contact( #PareggiatoreLong.DataOut.RestSolenoid )
      I_Contact( #PareggiatoreLong.DataIn.Work_Ls[1] )
      { S7_Templates := "time_type := Time" } #TON_Anticipi.Work.PareggLong.TON(pt := T#200MS, et =>)
   END_RUNG
   // the same network as SCL:
   #TON_Anticipi.Work.BattutaVrt.TON(IN := #BattutaVerticale.DataOut.WorkSolenoid AND NOT #BattutaVerticale.DataIn.Work_Ls[1],
                           PT := T#200MS);
   #TON_Anticipi.Work.PareggLong.TON(IN := #PareggiatoreLong.DataOut.RestSolenoid AND NOT #PareggiatoreLong.DataIn.Work_Ls[1],
                           PT := T#200MS);
END_REGION

REGION Network 4: Anticipi Movimento RIPOSO
   RUNG wire#powerrail
      Contact( #BattutaVerticale.DataOut.RestSolenoid )
      I_Contact( #BattutaVerticale.DataIn.Rest_Ls[1] )
      { S7_Templates := "time_type := Time" } #TON_Anticipi.Rest.BattutaVrt.TON(pt := T#200MS, et =>)
   END_RUNG
   RUNG wire#powerrail
      Contact( #PareggiatoreLong.DataOut.RestSolenoid )
      I_Contact( #PareggiatoreLong.DataIn.Rest_Ls[1] )
      { S7_Templates := "time_type := Time" } #TON_Anticipi.Rest.PareggLong.TON(pt := T#200MS, et =>)
   END_RUNG
   // the same network as SCL:
   #TON_Anticipi.Rest.BattutaVrt.TON(IN := #BattutaVerticale.DataOut.RestSolenoid AND NOT #BattutaVerticale.DataIn.Rest_Ls[1],
                           PT := T#200MS);
   #TON_Anticipi.Rest.PareggLong.TON(IN := #PareggiatoreLong.DataOut.RestSolenoid AND NOT #PareggiatoreLong.DataIn.Rest_Ls[1],
                           PT := T#200MS);
END_REGION

REGION Network 5: <+>
END_REGION

REGION Network 6: DataIn - FTC Input
   RUNG wire#powerrail
      Contact( #DataIn.Sens.FTC_Ingombro_In )
      { S7_Templates := "time_type := Time" } #IEC_FTC_Input.TON_Delay.TON(pt := #IEC_SP.FTC_Input.TON_PT, et =>)
   END_RUNG
   RUNG wire#powerrail
      Contact( #IEC_FTC_Input.TON_Delay.Q )
      { S7_Templates := "time_type := Time" } #IEC_FTC_Input.TOF_Delay.TOF(pt := #IEC_SP.FTC_Input.TOF_PT, et =>)
      Coil( #IEC_FTC_Input.FTC_On )
   END_RUNG
   // the same network as SCL:
   #IEC_FTC_Input.TON_Delay.TON(IN := #DataIn.Sens.FTC_Ingombro_In, PT := #IEC_SP.FTC_Input.TON_PT);
   #IEC_FTC_Input.TOF_Delay.TOF(IN := #IEC_FTC_Input.TON_Delay.Q, PT := #IEC_SP.FTC_Input.TOF_PT);
   #IEC_FTC_Input.FTC_On := #IEC_FTC_Input.TOF_Delay.Q;
END_REGION

REGION Network 7: DataIn - FTC Output
   RUNG wire#powerrail
      Contact( #DataIn.Sens.FTC_Ingombro_Out )
      { S7_Templates := "time_type := Time" } #IEC_FTC_Output.TON_Delay.TON(pt := #IEC_SP.FTC_Output.TON_PT, et =>)
   END_RUNG
   RUNG wire#powerrail
      Contact( #IEC_FTC_Output.TON_Delay.Q )
      { S7_Templates := "time_type := Time" } #IEC_FTC_Output.TOF_Delay.TOF(pt := #IEC_SP.FTC_Output.TOF_PT, et =>)
      Coil( #IEC_FTC_Output.FTC_On )
   END_RUNG
   // the same network as SCL:
   #IEC_FTC_Output.TON_Delay.TON(IN := #DataIn.Sens.FTC_Ingombro_Out, PT := #IEC_SP.FTC_Output.TON_PT);
   #IEC_FTC_Output.TOF_Delay.TOF(IN := #IEC_FTC_Output.TON_Delay.Q, PT := #IEC_SP.FTC_Output.TOF_PT);
   #IEC_FTC_Output.FTC_On := #IEC_FTC_Output.TOF_Delay.Q;
END_REGION

REGION Network 8: DataIn - FTC Presenza materiale
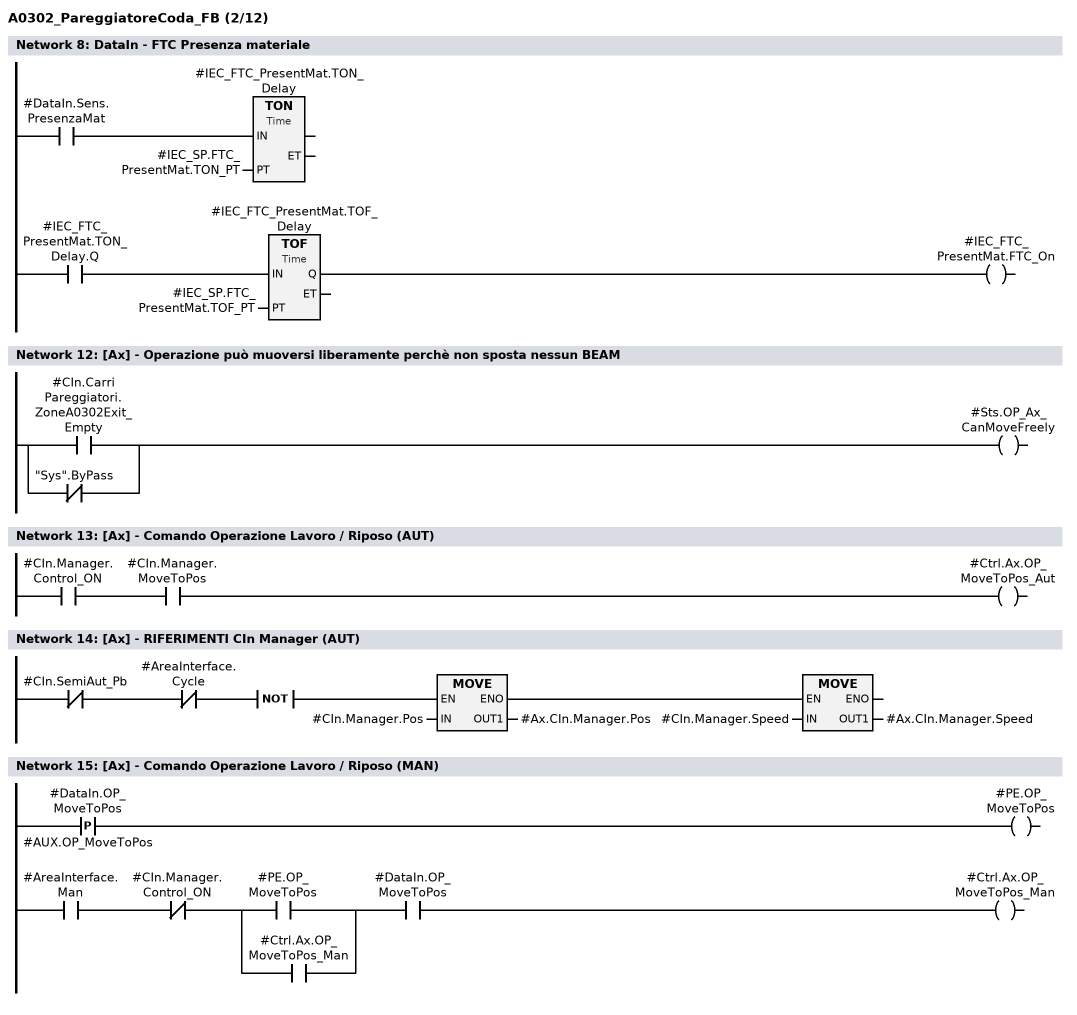
   RUNG wire#powerrail
      Contact( #DataIn.Sens.PresenzaMat )
      { S7_Templates := "time_type := Time" } #IEC_FTC_PresentMat.TON_Delay.TON(pt := #IEC_SP.FTC_PresentMat.TON_PT, et =>)
   END_RUNG
   RUNG wire#powerrail
      Contact( #IEC_FTC_PresentMat.TON_Delay.Q )
      { S7_Templates := "time_type := Time" } #IEC_FTC_PresentMat.TOF_Delay.TOF(pt := #IEC_SP.FTC_PresentMat.TOF_PT, et =>)
      Coil( #IEC_FTC_PresentMat.FTC_On )
   END_RUNG
   // the same network as SCL:
   #IEC_FTC_PresentMat.TON_Delay.TON(IN := #DataIn.Sens.PresenzaMat, PT := #IEC_SP.FTC_PresentMat.TON_PT);
   #IEC_FTC_PresentMat.TOF_Delay.TOF(IN := #IEC_FTC_PresentMat.TON_Delay.Q, PT := #IEC_SP.FTC_PresentMat.TOF_PT);
   #IEC_FTC_PresentMat.FTC_On := #IEC_FTC_PresentMat.TOF_Delay.Q;
END_REGION

REGION Network 9: <+>
END_REGION

REGION Network 10: <<< CARRO PAREGGIATORE CODA >>>
END_REGION

REGION Network 11: <+>
END_REGION

REGION Network 12: [Ax] - Operazione può muoversi liberamente perchè non sposta nessun BEAM
   RUNG wire#powerrail
      Contact( #CIn.CarriPareggiatori.ZoneA0302Exit_Empty )
      wire#w1
      Coil( #Sts.OP_Ax_CanMoveFreely )
   END_RUNG
   RUNG wire#powerrail
      I_Contact( "Sys".ByPass )
   END_RUNG wire#w1
   // the same network as SCL:
   #Sts.OP_Ax_CanMoveFreely := #CIn.CarriPareggiatori.ZoneA0302Exit_Empty OR NOT "Sys".ByPass;
END_REGION

REGION Network 13: [Ax] - Comando Operazione Lavoro / Riposo (AUT)
   RUNG wire#powerrail
      Contact( #CIn.Manager.Control_ON )
      Contact( #CIn.Manager.MoveToPos )
      Coil( #Ctrl.Ax.OP_MoveToPos_Aut )
   END_RUNG
   // the same network as SCL:
   #Ctrl.Ax.OP_MoveToPos_Aut := #CIn.Manager.Control_ON AND #CIn.Manager.MoveToPos;
END_REGION

REGION Network 14: [Ax] - RIFERIMENTI CIn Manager (AUT)
   RUNG wire#powerrail
      I_Contact( #CIn.SemiAut_Pb )
      I_Contact( #AreaInterface.Cycle )
      Not()
      Move(in := #CIn.Manager.Pos, out1 => #Ax.CIn.Manager.Pos)
      Move(in := #CIn.Manager.Speed, out1 => #Ax.CIn.Manager.Speed)
   END_RUNG
   // the same network as SCL:
   IF NOT (NOT #CIn.SemiAut_Pb AND NOT #AreaInterface.Cycle) THEN
       #Ax.CIn.Manager.Pos := #CIn.Manager.Pos;
       #Ax.CIn.Manager.Speed := #CIn.Manager.Speed;
   END_IF;
END_REGION

REGION Network 15: [Ax] - Comando Operazione Lavoro / Riposo (MAN)
   RUNG wire#powerrail
      P_Contact(operand := #DataIn.OP_MoveToPos, bit := #AUX.OP_MoveToPos)
      Coil( #PE.OP_MoveToPos )
   END_RUNG
   RUNG wire#powerrail
      Contact( #AreaInterface.Man )
      I_Contact( #CIn.Manager.Control_ON )
      wire#w1
      Contact( #PE.OP_MoveToPos )
      wire#w2
      Contact( #DataIn.OP_MoveToPos )
      Coil( #Ctrl.Ax.OP_MoveToPos_Man )
   END_RUNG
   RUNG wire#w1
      Contact( #Ctrl.Ax.OP_MoveToPos_Man )
   END_RUNG wire#w2
   // the same network as SCL:
   #_w1 := #DataIn.OP_MoveToPos AND NOT #AUX.OP_MoveToPos;   // rising edge of #DataIn.OP_MoveToPos
   #AUX.OP_MoveToPos := #DataIn.OP_MoveToPos;
   #PE.OP_MoveToPos := #_w1;
   #Ctrl.Ax.OP_MoveToPos_Man := #AreaInterface.Man AND NOT #CIn.Manager.Control_ON AND (#PE.OP_MoveToPos OR #Ctrl.Ax.OP_MoveToPos_Man) AND #DataIn.OP_MoveToPos;
END_REGION

REGION Network 16: <+>
END_REGION

